FUNCTION_BLOCK "COM_Modbus_CMV96"	// FB 1709
TITLE = Serial communication (Modbus to CMV)
//  
//COPYRIGHT:    (C) 1997 BY  BUHLER LTD.
//                           CH-9240 UZWIL  SWITZERLAND
//
//PRODUCT:      GCS90S7
//
//TITLE:        Modbus Interface to CMV96
//
//-------------------------------------------------------------------------
//
//IDENT:        AUTHOR:             DEPT:                       DATE:
//
//FB1707.1.0    A.Egli              CT3                         29-Mar-2004
//              1st Release in S7
//
//-------------------------------------------------------------------------
//
//PURPOSE:      MANUAL : see [COMxxMAN]
//
//RESTRICTIONS: S7
//
//-------------------------------------------------------------------------
//
AUTHOR : EA
FAMILY : GCS90LL
NAME : CVMModb
VERSION : 1.0
VAR_INPUT
  InComID : WORD  := W#16#1000;
  InTick200ms : BOOL ;	// Tick is every 200ms for one scan high
END_VAR
VAR
  Spare4 : INT ;
  ParRetryCnt : INT  := 1;
  ParTimeOut : INT  := 30;	//Timebase 0.1 s
  Spare10 : INT ;
  Spare12 : INT ;
  Spare14 : INT ;
  InIdx : INT ;
  InOutRestartTime : INT  := 50;	//Timebase 0.1 s
  OutMaxIdx : INT  := 5;
  OutLenDataRecord : INT  := 70;
  Error : STRUCT
   LCAddr : INT ;
   Status : INT ;
   Count : INT ;
   StatusSnd : INT ;
   StatusRcv : INT ;
   Spare0 : INT ;
   Spare2 : INT ;
   Spare3 : INT ;
  END_STRUCT ;
  Telegram : STRUCT
   Idx : INT ;	// Index of actual communication job
   LCAddr : INT ;	// Index of LC which data are send
   TimeOut : INT ;	//
   Step : INT ;
   RetryCnt : INT ;
   spare3 : INT ;
   spare4 : INT ;
   spare5 : INT ;
   spare6 : INT ;
   spare7 : INT ;
  END_STRUCT ;
  CVM0 : STRUCT
   InRead : BOOL ;	// Command to read data
   OutComFault : BOOL ;
   InAddr : INT ;
   ActivePower : DINT ;
   ReactivePowerInductive : DINT ;
   ReactivePowerCapacitive : DINT ;
   VoltageL1 : DINT ;
   CurrentL1 : DINT ;
   VoltageL2 : DINT ;
   CurrentL2 : DINT ;
   VoltageL3 : DINT ;
   CurrentL3 : DINT ;
   Spare40 : DINT ;
   Spare44 : DINT ;
   Spare48 : DINT ;
   Spare52 : DINT ;
   Spare56 : DINT ;
   Spare58 : DINT ;
   RetryCnt : INT ;
   tmpParaNr : INT ;
   Spare68 : INT ;
  END_STRUCT ;
  CVM : ARRAY  [1 .. 5 ] OF STRUCT
   InRead : BOOL ;	// Command to read data
   OutComFault : BOOL ;
   InAddr : INT ;
   ActivePower : DINT ;
   ReactivePowerInductive : DINT ;
   ReactivePowerCapacitive : DINT ;
   VoltageL1 : DINT ;
   CurrentL1 : DINT ;
   VoltageL2 : DINT ;
   CurrentL2 : DINT ;
   VoltageL3 : DINT ;
   CurrentL3 : DINT ;
   Spare40 : DINT ;
   Spare44 : DINT ;
   Spare48 : DINT ;
   Spare52 : DINT ;
   Spare56 : DINT ;
   Spare58 : DINT ;
   RetryCnt : INT ;
   Spare66 : INT ;
   Spare68 : INT ;
  END_STRUCT ;
  DataSnd : STRUCT
   Ident : BYTE ;
   Func : BYTE ;
   Data : ARRAY  [1 .. 20 ] OF INT ;
  END_STRUCT ;
  DataRcv : ARRAY  [0 .. 30 ] OF DINT ;
  BSND : SFB 12;	//Data of CFB =====
  BRCV : SFB 13;	//Data of LC
END_VAR
VAR_TEMP
  tmpstoreAR2 : DINT ;
  tmpAddrLC : DINT ;
  tmpNo : INT ;
  tmpRestart : BOOL ;
  tmpNext : BOOL ;
  tmpLoop2 : BOOL ;
END_VAR
BEGIN
NETWORK
TITLE = Store
      TAR2  #tmpstoreAR2;
NETWORK
TITLE = Call Siemens SFB
      NOP   0;
//-Receive--
      SET;
      S     #BRCV.EN_R;
      L     #Telegram.Step;
      L     2;
      ==I;
      A     #BRCV.NDR;
      JC    rsJ1;
      BLD   16;
      =     L 17.0;
      L     DINO;
      T     LW 15;
      CDB;
      OPN   DI [LW 15];
      TAR2  LD 11;
      L     DBW [AR2,P#0.0];
      T     #BRCV.ID;
//-Send--
      L     W#16#1002;
      T     DIW [AR2,P#684.0];
      L     124;
      T     DIW [AR2,P#686.0];
      L     DBNO;
      T     DIW [AR2,P#688.0];
      +AR2  P#522.0;
      TAR2;
      LAR2  LD 11;
      T     DID [AR2,P#690.0];
      +AR2  P#672.0;
      UC    "SIEMENS_BRCV";
      LAR2  LD 11;
      CDB;
      BLD   17;
rsJ1: BLD   16;
      =     L 17.0;
      L     DINO;
      T     LW 15;
      CDB;
      OPN   DI [LW 15];
      TAR2  LD 11;
      L     DBW [AR2,P#0.0];
      T     #BSND.ID;
      L     W#16#1002;
      T     DIW [AR2,P#658.0];
      L     42;
      T     DIW [AR2,P#660.0];
      L     DBNO;
      T     DIW [AR2,P#662.0];
      +AR2  P#480.0;
      TAR2;
      LAR2  LD 11;
      T     DID [AR2,P#664.0];
      +AR2  P#646.0;
      UC    "SIEMENS_BSEND";
      LAR2  LD 11;
      CDB;
      BLD   17;
NETWORK
TITLE = Methode 0: Control Step "Init" 
//===================================================
//====Init if Restart PLC ========
      L     0;
      L     #InOutRestartTime;
      <I;
      =     #tmpRestart;
      AN    #tmpRestart;
      JC    InJ0;
      L     0;
      T     #Error.Count;
      R     #BRCV.NDR;
      R     #BRCV.ERROR;
// Set send and receive buffer 
      AN    #InTick200ms;	// 200ms second pulse
      JC    sav0;
      L     #InOutRestartTime;
      +     -2;
      T     #InOutRestartTime;
      BEU;
InJ0: NOP   0;
NETWORK
TITLE = Step: 0 to 3: Read Element Data
// read element data of active element 
// this part is done for Step 1,2,3
      SET;
      R     #tmpNext;
      R     #tmpLoop2;
S0:   L     1;
      L     #Telegram.Idx;
      >I;
      JC    S0Nx;
      L     #OutMaxIdx;
      >I;
      JC    S0Nx;
      L     #Telegram.Idx;
      +     -1;
      L     #OutLenDataRecord;
      SLD   3;
      *I;
      L     P##CVM;
      +D;
      T     #tmpAddrLC;
      LAR1  #tmpAddrLC;
      LAR2  P##CVM0;
      L     D [AR1,P#0.0];
      T     D [AR2,P#0.0];
      L     D [AR1,P#4.0];
      T     D [AR2,P#4.0];
      L     D [AR1,P#8.0];
      T     D [AR2,P#8.0];
      L     D [AR1,P#12.0];
      T     D [AR2,P#12.0];
      L     D [AR1,P#16.0];
      T     D [AR2,P#16.0];
      L     D [AR1,P#20.0];
      T     D [AR2,P#20.0];
      L     D [AR1,P#24.0];
      T     D [AR2,P#24.0];
      L     D [AR1,P#28.0];
      T     D [AR2,P#28.0];
      L     D [AR1,P#32.0];
      T     D [AR2,P#32.0];
      L     D [AR1,P#36.0];
      T     D [AR2,P#36.0];
      L     D [AR1,P#40.0];
      T     D [AR2,P#40.0];
      L     D [AR1,P#44.0];
      T     D [AR2,P#44.0];
      L     D [AR1,P#48.0];
      T     D [AR2,P#48.0];
      L     D [AR1,P#52.0];
      T     D [AR2,P#52.0];
      L     D [AR1,P#56.0];
      T     D [AR2,P#56.0];
      L     D [AR1,P#60.0];
      T     D [AR2,P#60.0];
      L     D [AR1,P#64.0];
      T     D [AR2,P#64.0];
      L     W [AR1,P#68.0];
      T     W [AR2,P#68.0];
      LAR2  #tmpstoreAR2;
NETWORK
TITLE = Methode 0:  Control: Step "Test queue"
      L     0;
      L     #Telegram.Step;
      <>I;
      JC    S1;
//Second Loop
      A     #tmpNext;
      A     #CVM0.InRead;
      JC    xxS1;	//-->Send telegram
//--Search next element ----
S0Nx: L     1;
      L     #Telegram.Idx;
      +     1;
      T     #Telegram.Idx;
      >I;
      JC    S0X1;
      L     #OutMaxIdx;
      <=I;
      JC    S0Do;
//--First Element ---
S0X1: L     1;
      T     #Telegram.Idx;	//Init with Index 1
      A     #tmpLoop2;
      BEC;
      S     #tmpLoop2;
//--read element data ---
S0Do: S     #tmpNext;
      JU    S0;
NETWORK
TITLE = Methode Control: Transition to Step 1: Prepare Send Telegram
//Call back element control before send
xxS1: L     0;
      T     #Telegram.TimeOut;
      L     #CVM0.RetryCnt;
      T     #Telegram.RetryCnt;
//Start Telegram
      L     #CVM0.InAddr;
      T     #Telegram.LCAddr;
      T     #DataSnd.Ident;
      L     4;
      T     #DataSnd.Func;
//1st Register
      L     #CVM0.tmpParaNr;
      L     0;
      <>I;
      JC    RdJ1;
      L     20;
RdJ1: T     #DataSnd.Data[1];
      T     #CVM0.tmpParaNr;
//1st Number of register to read
      L     #DataSnd.Data[2];
      L     22;
      ==I;
      L     24;
      JC    S1J1;
      TAK;
S1J1: T     #DataSnd.Data[2];	//Number of register to read
//length of send data
      L     8;
      T     #BSND.LEN;
//Set address send buffer
//Send Next step
      L     1;	//-->Emptying Buffer
      T     #Telegram.Step;
      L     0;
      T     #Telegram.TimeOut;
//Send Next step
NETWORK
TITLE = Methode Control: Step1: Emptying buffer
S1:   L     #Telegram.Step;
      L     1;
      <>I;
      JC    S2;
// Wait one scan
      L     #BSND.STATUS;
      L     0;
      <>I;
      O     #BRCV.NDR;
      O     #BRCV.ERROR;
      O     #BSND.REQ;
      O     #BSND.ERROR;
      O     #BSND.DONE;
      O     #BSND.REQ;
      R     #BRCV.NDR;
      R     #BRCV.ERROR;
      R     #BSND.REQ;
      R     #BSND.ERROR;
      R     #BSND.DONE;
      R     #BSND.REQ;
      JC    sav0;
//------------------------------------
//Next Step  : Send Telegramm
      L     2;
      T     #Telegram.Step;
      L     0;
      T     #Telegram.TimeOut;
      SET;
      S     #BSND.REQ;
NETWORK
TITLE = Methode Control: Step 2 :Send telegram 
S2:   L     #Telegram.Step;
      L     2;
      <>I;
      JC    S3;
// Test telegram done         
      A     #BRCV.NDR;
      A     #BSND.DONE;
      JC    xxS3;
// Test Nak         
      A     #BSND.ERROR;
      L     #BSND.STATUS;
      JC    NAK;
// Test TimeOut         
      AN    #InTick200ms;
      JC    sav0;
      L     #Telegram.TimeOut;
      +     2;
      T     #Telegram.TimeOut;
      L     #ParTimeOut;
      >I;
      L     128;	// TimeOut 
      JC    NAK;	//--> Time out 
      JU    sav0;
NETWORK
TITLE = Methode Control: Step 3 : Test answer telegram
xxS3: NOP   0;
//====================================================
//Compare telegram lenght with requestet answer length
      L     #DataSnd.Data[2];	//Number of register to read
      L     2;
      *I;
      L     #BRCV.LEN;
      <>I;
      L     140;
      JC    NAK;
//====================================================
//Store Data
      L     0;
      L     #DataSnd.Data[1];
      <>I;
      JC    AWJ1;
      L     #DataRcv[0];
      T     #CVM0.VoltageL1;
      L     #DataRcv[1];
      T     #CVM0.CurrentL1;
      L     #DataRcv[5];
      T     #CVM0.VoltageL2;
      L     #DataRcv[6];
      T     #CVM0.CurrentL2;
      L     #DataRcv[10];
      T     #CVM0.VoltageL3;
      L     #DataRcv[11];
      T     #CVM0.CurrentL3;
AWJ1: L     20;
      L     #DataSnd.Data[1];
      <>I;
      JC    AWJ9;
      L     #DataRcv[0];
      T     #CVM0.VoltageL3;
      L     #DataRcv[1];
      T     #CVM0.CurrentL3;
      L     #DataRcv[5];
      T     #CVM0.ActivePower;
      L     #DataRcv[6];
      T     #CVM0.ReactivePowerInductive;
      L     #DataRcv[7];
      T     #CVM0.ReactivePowerCapacitive;
AWJ9: SET;
      R     #CVM0.OutComFault;
NETWORK
TITLE = Methode Control: Step 3: Init for next Telegram
S3:   L     0;
      T     #CVM0.RetryCnt;
S3rt: SET;
      R     #BRCV.NDR;
      R     #BRCV.ERROR;
      R     #BSND.DONE;
      R     #BSND.ERROR;
//--Step 0 -----
      L     0;
      T     #Telegram.Step;
      JU    sav0;
NETWORK
TITLE = Methode Control: NAK 
///
//Error send 
NAK:  T     #Error.Status;
      L     #Telegram.LCAddr;
      T     #Error.LCAddr;
      L     #Error.Count;
      +     1;
      T     #Error.Count;
      L     #BSND.STATUS;
      T     #Error.StatusSnd;
      L     #BRCV.STATUS;
      T     #Error.StatusRcv;
      L     #ParRetryCnt;
      L     #CVM0.RetryCnt;
      >I;	//--> Retry after fault 
      O     #tmpRestart;	//--> Retry during restart
      JC    naRt;	//--> Retry after fault 
      L     0;
      T     #CVM0.RetryCnt;
      S     #CVM0.OutComFault;
      JU    S3;
naRt: L     #CVM0.RetryCnt;
      +     1;
      T     #CVM0.RetryCnt;
      JU    S3rt;
NETWORK
TITLE = Methode 2: Store element data 
sav0: L     1;
      L     #Telegram.Idx;
      >I;
      BEC;
      L     #OutMaxIdx;
      >I;
      BEC;
      L     #Telegram.Idx;
      +     -1;
      L     #OutLenDataRecord;
      SLD   3;
      *I;
      L     P##CVM;
      +D;
      T     #tmpAddrLC;
      LAR1  P##CVM0;
      LAR2  #tmpAddrLC;
      L     D [AR1,P#0.0];
      T     D [AR2,P#0.0];
      L     D [AR1,P#4.0];
      T     D [AR2,P#4.0];
      L     D [AR1,P#8.0];
      T     D [AR2,P#8.0];
      L     D [AR1,P#12.0];
      T     D [AR2,P#12.0];
      L     D [AR1,P#16.0];
      T     D [AR2,P#16.0];
      L     D [AR1,P#20.0];
      T     D [AR2,P#20.0];
      L     D [AR1,P#24.0];
      T     D [AR2,P#24.0];
      L     D [AR1,P#28.0];
      T     D [AR2,P#28.0];
      L     D [AR1,P#32.0];
      T     D [AR2,P#32.0];
      L     D [AR1,P#36.0];
      T     D [AR2,P#36.0];
      L     D [AR1,P#40.0];
      T     D [AR2,P#40.0];
      L     D [AR1,P#44.0];
      T     D [AR2,P#44.0];
      L     D [AR1,P#48.0];
      T     D [AR2,P#48.0];
      L     D [AR1,P#52.0];
      T     D [AR2,P#52.0];
      L     D [AR1,P#56.0];
      T     D [AR2,P#56.0];
      L     D [AR1,P#60.0];
      T     D [AR2,P#60.0];
      L     D [AR1,P#64.0];
      T     D [AR2,P#64.0];
      L     W [AR1,P#68.0];
      T     W [AR2,P#68.0];
      LAR2  #tmpstoreAR2;
END_FUNCTION_BLOCK

FUNCTION_BLOCK "SSA_EL_Sampler_RFID"	// FB 1714
TITLE = Lesen/Schreiben 2k bit / Profibus DP
//COPYRIGHT:    (C) 2006  BUHLER AG, CH-9240 UZWIL, SWITZERLAND
//
//PRODUCT:      GCS7R2
//
//TITLE:        RFID Baumer
//
//REVISION:     20
//-------------------------------------------------------------------------
//
//IDENT:        AUTHOR:             DEPT:                       DATE:
//FB1714.1.0    A. Egli             CT3                         12-Sep-2007
//              #FromBuhler.InSimulation to read/write process immage
//FB1714.1.0    A. Egli             CT3                         19-Mar-2007
//              New Release R2
//
//-------------------------------------------------------------------------
//
//PURPOSE:      MANUAL : see [SSW-EL-Sampler_MAN_en]
//              This FB is a copy of original communication block FB102 of 
//              Baumer. 
//
//              Modification of BUHLER:
//              - Move all IN and OUT signal to the area STAT.
//              - Add all data of the global DB of Baumer into are STAT
//                (STAT:IN,STAT:OUT)
//                The structur IN must start at Byte 0
//                The structur OUT must start at Byte 204
//                This because Baumer uses the absoulte address of thes tags
//             - Add interface to BUHLER elements
//               (FromBuhler, ToBuhler)  
//              
//
//RESTRICTIONS: S7
//
//-------------------------------------------------------------------------
//
AUTHOR : ZIEGERT
FAMILY : BAUMER
NAME : RFID
VERSION : 1.1
VAR
  IN : STRUCT 	//Read buffer
   CONTROL1 : WORD ;	//Commando / # antenne
   CONTROL2 : WORD ;	//State of central unit / # pages
   CONTROL3 : WORD ;	//# datablocks / Actual datablock
   CONTROL4 : WORD ;	//Length of datablock / Controlbyte
   PAGE16 : DWORD ;	//Nutzdaten 1 Input
   PAGE17 : DWORD ;	//Nutzdaten 2 Input
   PAGE18 : DWORD ;	//Nutzdaten 3 Input
   PAGE19 : DWORD ;	//Nutzdaten 4 Input
   PAGE20 : DWORD ;	//Nutzdaten 5 Input
   PAGE21 : DWORD ;	//Nutzdaten 6 Input
   PAGE22 : DWORD ;	//Nutzdaten 7 Input
   PAGE23 : DWORD ;	//Nutzdaten 8 Input
   PAGE24 : DWORD ;	//Nutzdaten 9 Input
   PAGE25 : DWORD ;	//Nutzdaten 10 Input
   PAGE26 : DWORD ;	//Nutzdaten 11 Input
   PAGE27 : DWORD ;	//Nutzdaten 12 Input
   PAGE28 : DWORD ;	//Nutzdaten 13 Input
   PAGE29 : DWORD ;	//Nutzdaten 14 Input
   PAGE30 : DWORD ;	//Nutzdaten 15 Input
   PAGE31 : DWORD ;	//Nutzdaten 16 Input
   PAGE32 : DWORD ;	//Nutzdaten 17 Input
   PAGE33 : DWORD ;	//Nutzdaten 18 Input
   PAGE34 : DWORD ;	//Nutzdaten 19 Input
   PAGE35 : DWORD ;	//Nutzdaten 20 Input
   PAGE36 : DWORD ;	//Nutzdaten 21 Input
   PAGE37 : DWORD ;	//Nutzdaten 22 Input
   PAGE38 : DWORD ;	//Nutzdaten 23 Input
   PAGE39 : DWORD ;	//Nutzdaten 24 Input
   PAGE40 : DWORD ;	//Nutzdaten 25 Input
   PAGE41 : DWORD ;	//Nutzdaten 26 Input
   PAGE42 : DWORD ;	//Nutzdaten 27 Input
   PAGE43 : DWORD ;	//Nutzdaten 28 Input
   PAGE44 : DWORD ;	//Nutzdaten 29 Input
   PAGE45 : DWORD ;	//Nutzdaten 30 Input
   PAGE46 : DWORD ;	//Nutzdaten 31 Input
   PAGE47 : DWORD ;	//Nutzdaten 32 Input
   PAGE48 : DWORD ;	//Nutzdaten 33 Input
   PAGE49 : DWORD ;	//Nutzdaten 34 Input
   PAGE50 : DWORD ;	//Nutzdaten 35 Input
   PAGE51 : DWORD ;	//Nutzdaten 36 Input
   PAGE52 : DWORD ;	//Nutzdaten 37 Input
   PAGE53 : DWORD ;	//Nutzdaten 38 Input
   PAGE54 : DWORD ;	//Nutzdaten 39 Input
   PAGE55 : DWORD ;	//Nutzdaten 40 Input
   PAGE56 : DWORD ;	//Nutzdaten 41 Input
   PAGE57 : DWORD ;	//Nutzdaten 42 Input
   PAGE58 : DWORD ;	//Nutzdaten 43 Input
   PAGE59 : DWORD ;	//Nutzdaten 44 Input
   PAGE60 : DWORD ;	//Nutzdaten 45 Input
   PAGE61 : DWORD ;	//Nutzdaten 46 Input
   PAGE62 : DWORD ;	//Nutzdaten 47 Input
   PAGE63 : DWORD ;	//Nutzdaten 48 Input
   Spare : DWORD ;	//spare
  END_STRUCT ;
  OUT : STRUCT 	//Write buffer
   CONTROL1 : WORD ;	//Commando / # antenne
   CONTROL2 : WORD ;	//Startpage / # pages
   CONTROL3 : WORD ;	//# datablocks / Actual datablock
   CONTROL4 : WORD ;	//Length of datablock / Controlbyte
   PAGE16 : DWORD ;	//Nutzdaten 1 Output
   PAGE17 : DWORD ;	//Nutzdaten 2 Output
   PAGE18 : DWORD ;	//Nutzdaten 3 Output
   PAGE19 : DWORD ;	//Nutzdaten 4 Output
   PAGE20 : DWORD ;	//Nutzdaten 5 Output
   PAGE21 : DWORD ;	//Nutzdaten 6 Output
   PAGE22 : DWORD ;	//Nutzdaten 7 Output
   PAGE23 : DWORD ;	//Nutzdaten 8 Output
   PAGE24 : DWORD ;	//Nutzdaten 9 Output
   PAGE25 : DWORD ;	//Nutzdaten 10 Output
   PAGE26 : DWORD ;	//Nutzdaten 11 Output
   PAGE27 : DWORD ;	//Nutzdaten 12 Output
   PAGE28 : DWORD ;	//Nutzdaten 13 Output
   PAGE29 : DWORD ;	//Nutzdaten 14 Output
   PAGE30 : DWORD ;	//Nutzdaten 15 Output
   PAGE31 : DWORD ;	//Nutzdaten 16 Output
   PAGE32 : DWORD ;	//Nutzdaten 17 Output
   PAGE33 : DWORD ;	//Nutzdaten 18 Output
   PAGE34 : DWORD ;	//Nutzdaten 19 Output
   PAGE35 : DWORD ;	//Nutzdaten 20 Output
   PAGE36 : DWORD ;	//Nutzdaten 21 Output
   PAGE37 : DWORD ;	//Nutzdaten 22 Output
   PAGE38 : DWORD ;	//Nutzdaten 23 Output
   PAGE39 : DWORD ;	//Nutzdaten 24 Output
   PAGE40 : DWORD ;	//Nutzdaten 25 Output
   PAGE41 : DWORD ;	//Nutzdaten 26 Output
   PAGE42 : DWORD ;	//Nutzdaten 27 Output
   PAGE43 : DWORD ;	//Nutzdaten 28 Output
   PAGE44 : DWORD ;	//Nutzdaten 29 Output
   PAGE45 : DWORD ;	//Nutzdaten 30 Output
   PAGE46 : DWORD ;	//Nutzdaten 31 Output
   PAGE47 : DWORD ;	//Nutzdaten 32 Output
   PAGE48 : DWORD ;	//Nutzdaten 33 Output
   PAGE49 : DWORD ;	//Nutzdaten 34 Output
   PAGE50 : DWORD ;	//Nutzdaten 35 Output
   PAGE51 : DWORD ;	//Nutzdaten 36 Output
   PAGE52 : DWORD ;	//Nutzdaten 37 Output
   PAGE53 : DWORD ;	//Nutzdaten 38 Output
   PAGE54 : DWORD ;	//Nutzdaten 39 Output
   PAGE55 : DWORD ;	//Nutzdaten 40 Output
   PAGE56 : DWORD ;	//Nutzdaten 41 Output
   PAGE57 : DWORD ;	//Nutzdaten 42 Output
   PAGE58 : DWORD ;	//Nutzdaten 43 Output
   PAGE59 : DWORD ;	//Nutzdaten 44 Output
   PAGE60 : DWORD ;	//Nutzdaten 45 Output
   PAGE61 : DWORD ;	//Nutzdaten 46 Output
   PAGE62 : DWORD ;	//Nutzdaten 47 Output
   PAGE63 : DWORD ;	//Nutzdaten 48 Output
   PAGE64 : DWORD ;	//Nutzdaten 49 Output
  END_STRUCT ;
  spare408 : BOOL ;
  FromBuhler : STRUCT
   BottleInPosition : BOOL ;	//LS tells that a bottle is in position
   StBottleChange : BOOL ;	//Bottle change is avtive
   CmdFaultReset : BOOL ;	//Reset Retry Counter
   ParTag2KB : BOOL ;	//1=2kByte  , 0=256Byte
   InSimulation : BOOL ;	//1=Connected to IOSimuli
   ParByteNo : INT ;	//1st Byte of ID
   spare1 : INT ;
   spare2 : INT ;
   spare3 : INT ;
  END_STRUCT ;
  ToBuhler : STRUCT
   OutReadingFault : BOOL ;
   RFIDJobRunning : BOOL ;	//Data for user
   EdgeBottleInPossition : BOOL ;	//Data for user
   RFIDStartReading : BOOL ;	//Data for user
   OutEdgeBreak : BOOL ;
   OutEdgeRW_End : BOOL ;
   OutPulseRW_End : BOOL ;
   OutRFIDBusy : BOOL ;
   OutEdgeRFIDIdling : BOOL ;
   OutPulseRFIDIdling : BOOL ;
   OutRFIDIdling : BOOL ;
   OutTimeOut : INT ;
   OutTagNoAct : DINT ;
   OutDelayBrake : INT ;
   OutRetryCounter : INT ;
   spare1 : INT ;
   spare2 : INT ;
   spare3 : INT ;
   spare4 : INT ;
   spare5 : INT ;
  END_STRUCT ;
  START_RW : BOOL ;	//Start read/write Auftrag
  BREAK : BOOL ;	//Break read/write
  READ : BOOL ;	//Commando read
  WRITE : BOOL ;	//Commando write
  POLL : BOOL ;	//Mode poll
  AUTO : BOOL ;	//Mode automatic
  CONT : BOOL ;	//Mode continues
  ANT : INT ;	//Nr. der Antenne (Wert 0-2)
  STARTP : INT ;	//Startpage (Wert >=16, <=48)
  ANZP : INT ;	//Anzahl Page Extern (Wert = 1-48)
  EA_or_PW : INT ;	//Vorwahl Adressbereich E/A oder PW, (Wert 0 = E/A Wert 1 = PW)
  EADR : INT ;	//Anfangsaddresse Eingänge (Daten vom slave)
  AADR : INT ;	//Anfangsaddresse Ausgänge (Daten vom slave)
  T_MS : INT ;	//Zeitwert für Time out
  STATE_HW : BYTE ;	//Status des OIS-L Controller's (read/write system)
  STATE_HS : BYTE ;	//Status handshake
  RW_END : BOOL ;	//Read/Write Ende
  TIMEOUT : BOOL ;	//Timeout
  PARA : BOOL ;	//Parameterfehler
  FLT : BOOL ;	//Sammelfehler
  HW_FLT : BOOL ;	//Hardware Fehler OIS-L Controller
  P_start_rw : BOOL ;	//Flanke 'START_RW'
  E_start_rw : BOOL ;	//Hilfsmerker 'START_RW'
  RW_act : BOOL ;	//Auftrag gestartet
  P_rw_end : BOOL ;	//Pos. Flanke Lese/schreiben ende
  E_rw_end : BOOL ;	//Enable Flanke Lesen/schreiben Ende
  ANZP_SAVE : INT ;	//Pageanzahl sichern
  anz_page : INT ;	//Anzahl Page intern (wert = 0-15)
  anz_blocks : INT ;	//# Anzahl Datenblocks
  act_block : INT ;	//# Write: Aktueller Datenblock
  rest_bytes : INT ;	//# Anzahl Restbyte's die ggelesen/geschrieben werden
  anz_bytes : INT ;	//# Anzahl Byt's gesamt
  rcv_blocks : INT ;	//# Aktueller Blockzeiger
  P_OIS_new_data : BOOL ;	//# Read: Flanke start neue Daten Lesen
  E_OIS_new_data : BOOL ;	//# Read: Hilfsmerker: neue Daten Lesen
  P_OIS_data_rcv : BOOL ;	//# Write: Flanke start neue Daten Schreiben
  E_OIS_data_rcv : BOOL ;	//# Write: Hilfsmerker: neue Date Schreiben
  RD : BOOL ;	//# Read: Start Daten Lesen
  RD_no_active : BOOL ;	//# Read/Write: Daten Lesen/Schreiben nicht active
  WR : BOOL ;	//# Write: Start Daten Schreiben
  pointer_dest : DWORD ;	//Pointer Hilfsregister zum zwischenspeichern des Zeigers
  Pointer_buffer : DWORD ;	//Pointer aktueller Zeiger auf Daten/Adressbereich
  s_pointer_set : BOOL ;	//Pointer_buffer gesetzt
  S_break : BOOL ;	//positive Flanke Breakbefehl gestartet
  E_break : BOOL ;	//Flankenmerker Break
  N_break : BOOL ;	//negative Flanke nach S_break, Break an OIS-L senden
  S_poll : BOOL ;	//Mode poll angewählt
  E_en_poll : BOOL ;	//Hilfsmerker poll angewählt
  S_auto : BOOL ;	//Mode auto angewählt
  E_en_auto : BOOL ;	//Hilfsmerker auto angewählt
  S_cont : BOOL ;	//Mode cont angewählt
  E_en_cont : BOOL ;	//Hilfsmerker cont angewählt
  anz_loop : INT ;	//# Read/Write: Anzahl der errechneten loop's
  Loop : INT ;	//Schleife für mehrfachse Lesen (Wert 0-2)
  S_loop : BOOL ;	//Schleifenmerker (1 wenn mehr als 16 Page gelesen werden sollen)
  S_Data_1 : BOOL ;	//Berechnung für Startpage und Anzahl Page durchgeführt
  E_en_Bussy : BOOL ;	//Auftrag gestartet
  P_en_DATA : BOOL ;	//Hilfsmerker pos.Flanke: neue daten vom Slave vorhanden
  N_en_DATA : BOOL ;	//Hilfsmerker neg.Flanke: neue daten vom Slave vorhanden
  E_en_DATA : BOOL ;	//Flanke neue Daten vom Slave vorhanden
  adb_dbn : BOOL ;	//# Read/Write: Controll In ADB = DBN
  errCDO : BOOL ;	//Fehler
  errMOD : BOOL ;	//Fehler Mode Read/Write (beide angewählt)
  errANT : BOOL ;	//Fehler Nr. der Antenne (darf nur 1 oder 2 sein)
  errSTARTP : BOOL ;	//Fehler Startpage (min Wert 16, max Wert 63)
  errANZP : BOOL ;	//Fehler Anzahl Page {min Wert 1, max Wert 48 (cont mode max 16)}
  errDATA : BOOL ;	//Fehler Datenlänge und Controllbit CTL.0 und CTL.2
  E_CTL_7_out : BOOL ;	//Flankenmerker CTL.7 out
  s_timeout : BOOL ;	//Start Timeout bei CLT(out)<> CLT(in)
  s_daten_ok : BOOL ;	//Daten liegen auf den Ausgängen (write)
  s_next_block : BOOL ;	//Daten an oil-s, nächsten Block senden
  dummy : BOOL ;	//Schmiermerker
  result : INT ;	//Hilfsregister: Check Anzahl page
  rest_page : INT ;	//Register: dient zum zwischenspeichern der neu ermittelten Pageanzahl
  Pointer_input : DWORD ;	//Pointer input: Zeiger auf Eingangsbereich
  Pointer_output : DWORD ;	//Pointer output: Zeiger auf Ausgangsbereich
  RD_loop_counter : INT ;	//#Read/Write: Schleifenzähler beim Lesen und Schreiben
END_VAR
VAR_TEMP
  tmpDB : INT ;
  tmpTOut : INT ;
END_VAR
BEGIN
NETWORK
TITLE =
//Dieser FB ist die Schnittstelle für das Lesen und Schreiben von 2k Tag's über 
//den Profibus DP vom oder zum OIS-L Kontroller.
//Folgende Funktionen können mit dem FB realiesiert werden:
//Lesen von 48 Page im Poll und Auto Mode
//Lesen von 16 Page im Cont Mode
//Schreiben von 48 Page im Poll und Auto Mode
//Das Schreiben im Cont Mode ist nicht möglich.
//--------------------------------------------------------------------------------
//Die Beschreibung der einzelnen Modis ist dem Benutzerhandbuch für den OIS-L 
//Kontroller zu entnehmen.
//--------------------------------------------------------------------------------
//Datenstruktur im _DB
//DB102--------------------
//DBW0  Comando/Antenne                      [IN]
//DBW2  Status/AnzPage                       [IN]
//DBW4  AnzDatenblöcke/Nr.Akt.Datenblock     [IN]
//DBW6  Datenlänge/Controllbyte              [IN]
//DD8-DD196  Daten Page 16-63                [IN]
//
//DBW204 Comando/Antenne                     [OUT]
//DBW206 Status/AnzPage                      [OUT]
//DBW208 AnzDatenblöcke/Nr.Akt.Datenblock    [OUT]
//DBW210 Datenlänge/Controllbyte             [OUT]
//DD212-DD400 Daten Page 16-63               [OUT]
//
//Achtung: Der Datenbereich für Daten von Antenne 1 und Daten von Antenne 2 sind 
//identisch.  Alternativ können auch bei einem Mehrfachaufruf zwei Datenbausteine 
//eingesetzt werden, in denen die Tag-Daten abgespeichert werden.
//Bei Mehrfachaufrufen ist darauf zu achten, das bevor der FB durchlaufen wird 
//ein Break Befehl durchgeführt wird.
//
//Weiterhin ist darauf zu achten, dass die FB's gegeneinander Verriegelt werden.
//Ein Möglichkeit ist es durch die Anwahl der Antennen den EN Eingang der FB's zu 
//selktieren und das RD_End Signal als Quittierung zu benutzen.
//
//Continius-Mode:
//Nach einem Break-Befehl während des Continius-Mode muß erneut ein Startbefehl 
//abgesetzt werden um das Lesen zu starten:
//
//Zusätzlich benötig der FB noch einen Instanz DB, der beim Aufruf des FB's 
//eingetragen werden muß. Es ist nicht empfehlenswert den FB105 in eine 
//Multiinstanz abzuändern.
//
//Parameterbeschreibung:
//---------EINGÄNGE----------
//EN       [Bool]     Enable muß auf Logisch 1 sein.
//_DB      [Bloch_DB] Datenbaustein der die Tagdaten sowie Status-und Steuerwort  
//                    enthält.
//START_RD [Bool]     Daten lesen start im Poll- und Auto-Mode.
//BREAK    [Bool]     Hi aktiv, setzt den IBS-OISL-Protokollkoppler
//POLL     [Bool]     Hi aktiv Pollmodus.
//AUTO     [Bool]     Hi aktiv Automatikmodus.
//CONT     [Bool]     Hi aktiv Continiusmode.
//READ     [Bool]     Hi aktiv selektiert den Lesevorgang
//WRITE    [Bool]     Hi aktiv selektiert den Schreibvorgang 
//ANT      [Int]      Wert 1 oder 2 aktiviert den Anteneneingang 1 oder 2.
//STARTP   [INT]      Wert 16-63 Vorwahl der Page, ab der Daten gelesen oder
//                    beschrieben werden sollen
//ANZP     [INT]      Wert 1-48 Anzahl Page's die gelesen oder beschrieben werden 
//                    sollen {max. 48 Page's können gelesen oder beschrieben 
//                    werden, im cont Mode ist das lesen auf 16 Page reduziert}.
//EA_or_PW [Int]      Ermöglicht die Anpassung des Einganmgsbereichs Wert 0=EA,   
//                    Wert 1=PW (PW = Peripheriebereich)
//EADR     [Int]      Wert je nach parametrierten Eingangsbereich Profibus/S7.
//AADR     [Int]      Wert je nach parametrierten Eingangsbereich Profibus/S7.
//T_OUT    [Timer]    S7 Zeit (z.B. T10) Überwachung der Lesefunktion im 
//                    AUTO-CONT-Mode.
//T_OUT_MS [S5Time]   Zeitbereich von T_OUT (z.B. S5T#10s).
//
//---------AUSGÄNGE----------
//ENO      [Bool]     Logisch 1 wenn EN Logisch 1 ist.
//STATE_HW [Byte]     Status und Errocode des OISL-Protokollkoppler.
//State_HS [Byte]     Status Controllbyts des OISL-Protokollkoppler.
//RD_END   [Bool]     Hi aktiv, Lese/Schreib-Auftrag beendet.
//TIMEOUT  [Bool]     Hi aktiv, Zeitüberschreitung beim lesen (kein Tag im        
//                    Antennenbereich).
//PARA     [Bool]     Hi aktiv, Falsche Parameter an den Eingängen POLL, AUTO,CONT
//                    oder ANT.
//FLT      [Bool]     Hi aktiv, Summenfehler.
//
//Beschreibung zum Ablauf:
//Liegt an den Eingängen (Poll, Auto, Cont oder Antenne) kein Singnal wird der 
//Ausgang PARA und FTL gesetzt und zum Ende verzweigt.
//Nachdem ein Modus gewählt wurde kann das Lesen/Schreiben der Daten mit START_RD 
//eingeleitet werden. Ein beschreiben der Tag's im Continus-Mode ist nicht 
//möglich.
//Wurde ein Modus vorgewählt und das Lesen der Daten gestartet, sollte bei einem 
//wechsel des Modus immer ein Reset Buffer durchgeführt werden.
//Im Auto/Cont Mode ist die Zeitüberwachung aktiv im Poll Mode nicht.
//Im Cont_Mode führt eine Pageanzahl >16 zum setzten des Fehlerausgangs.
//Ein Break-Befehl kann nur bei eindeutiger Parametrierung am Eingang 
//durchgeführt werden.
//Wird als StartPage 0 und AnzahlPage 1 vorgegeben, wird die TAG ID ausgelesen. 
//
NETWORK
TITLE = [1.0] öffen _DB 
      L     DINO;
      T     #tmpDB;
      OPN   DB [#tmpDB];
NETWORK
TITLE = [1.0] BUZ: Command from Buhler to Baumer RFID (Part 1)
      NOP   0;
//-Initialize ---
      AN    DIX 442.2;
      S     DIX 442.2;
      S     DIX 442.1;
// 
//-Reading---
      A     DIX 410.0;
      AN    DIX 410.2;
      FP    DIX 420.2;
      S     DIX 420.3;
// 
      A     DIX 420.3;
      AN    DIX 420.7;
      A     DIX 421.2;
      AN    DIX 442.1;
      S     DIX 442.0;
//WinTrend      L     S5T#150MS
//WinTrend      SV    T    200
//WinTrend      U     T    200
//WinTrend      =     M   1400.0
// 
      O     DIX 410.1;
      R     DIX 420.3;
// 
//-Set default data---
      SET;
      R     DIX 442.3;
      S     DIX 442.4;
      R     DIX 442.5;
      R     DIX 442.6;
      L     0;	//[1.1]
      A     DIX 410.4;	//[1.1]
      JC    SiEA;	//[1.1]
      L     1;
SiEA: T     DIW 450;
      L     1;
      T     DIW 444;
      L     0;
      T     DIW 446;
      L     1;
      T     DIW 448;
      L     DIW 412;
      T     DIW 452;
      L     DIW 412;
      T     DIW 454;
      L     2000;
      T     DIW 456;
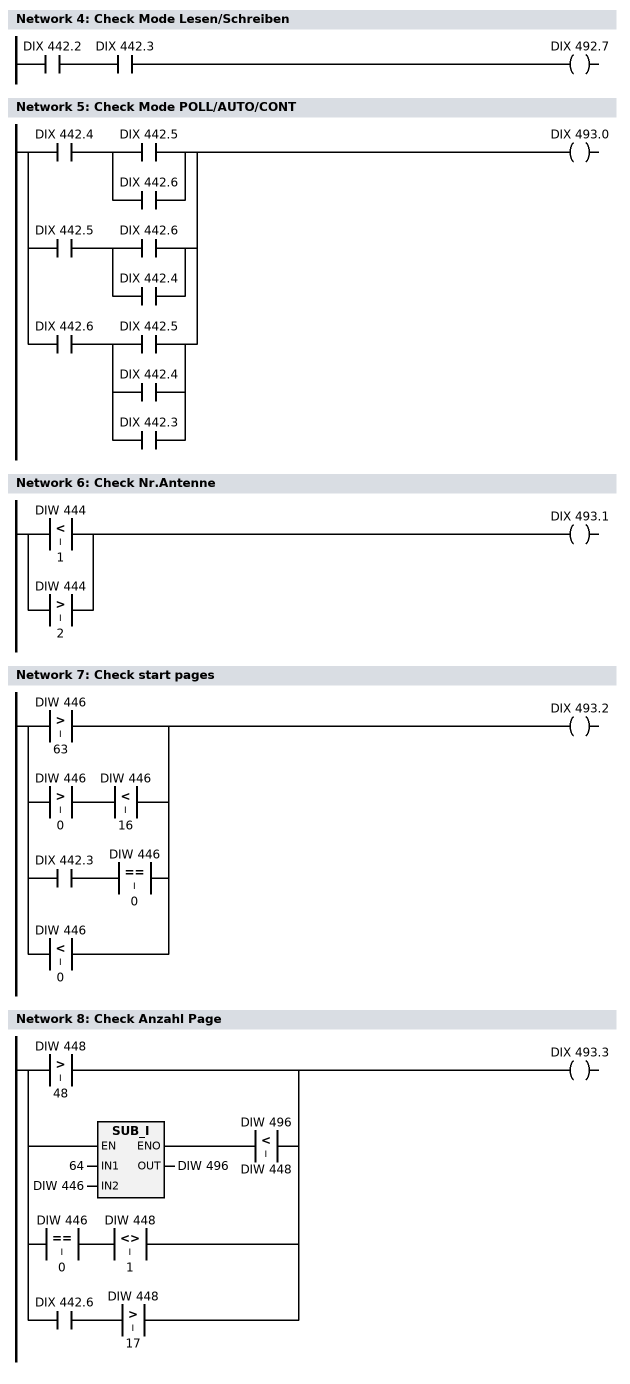
NETWORK
TITLE = Check Mode Lesen/Schreiben
      A     DIX 442.2;
      A     DIX 442.3;
      =     DIX 492.7;
NETWORK
TITLE = Check Mode POLL/AUTO/CONT
      A     DIX 442.4;
      A(;
      O     DIX 442.5;
      O     DIX 442.6;
      );
      O;
      A     DIX 442.5;
      A(;
      O     DIX 442.6;
      O     DIX 442.4;
      );
      O;
      A     DIX 442.6;
      A(;
      O     DIX 442.5;
      O     DIX 442.4;
      O     DIX 442.3;
      );
      =     DIX 493.0;
NETWORK
TITLE = Check Nr.Antenne
      O(;
      L     DIW 444;
      L     1;
      <I;
      );
      O(;
      L     DIW 444;
      L     2;
      >I;
      );
      =     DIX 493.1;
NETWORK
TITLE = Check start pages
      O(;
      L     DIW 446;
      L     63;
      >I;
      );
      O;
      A(;
      L     DIW 446;
      L     0;
      >I;
      );
      A(;
      L     DIW 446;
      L     16;
      <I;
      );
      O;
      A     DIX 442.3;
      A(;
      L     DIW 446;
      L     0;
      ==I;
      );
      O(;
      L     DIW 446;
      L     0;
      <I;
      );
      =     DIX 493.2;
NETWORK
TITLE = Check Anzahl Page
      O(;
      L     DIW 448;
      L     48;
      >I;
      );
      O(;
      A(;
      L     64;
      L     DIW 446;
      -I;
      T     DIW 496;
      AN    OV;
      SAVE;
      CLR;
      A     BR;
      );
      A(;
      L     DIW 496;
      L     DIW 448;
      <I;
      );
      );
      O;
      A(;
      L     DIW 446;
      L     0;
      ==I;
      );
      A(;
      L     DIW 448;
      L     1;
      <>I;
      );
      O;
      A     DIX 442.6;
      A(;
      L     DIW 448;
      L     17;
      >I;
      );
      =     DIX 493.3;
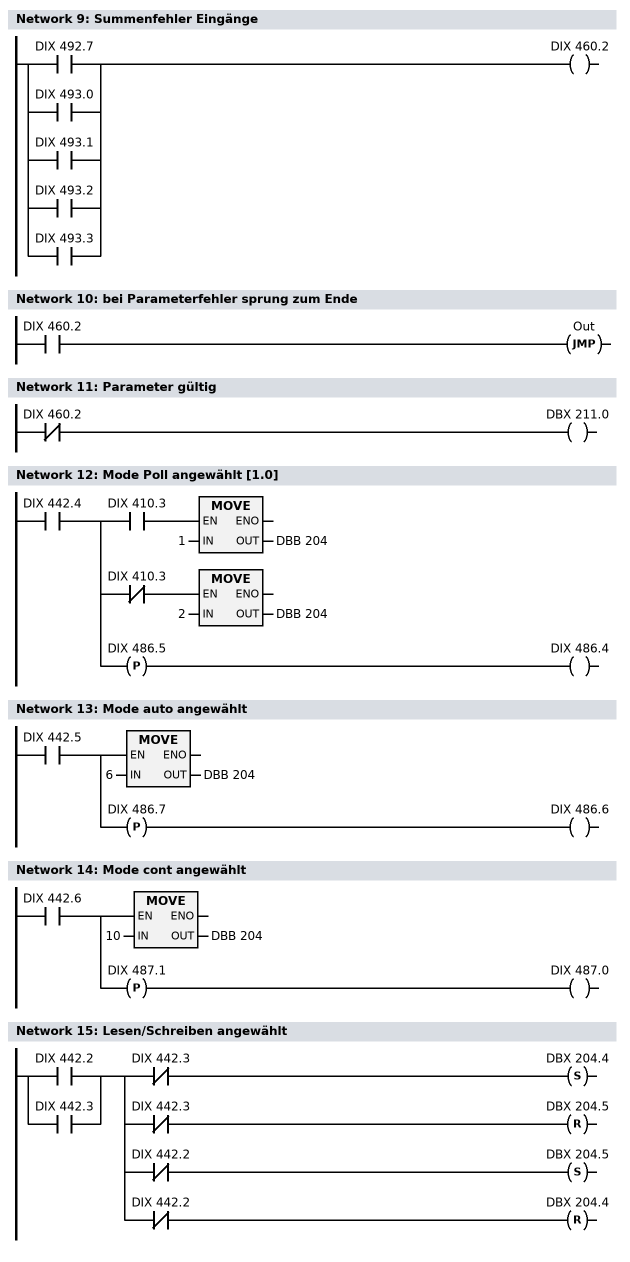
NETWORK
TITLE = Summenfehler Eingänge
      O     DIX 492.7;
      O     DIX 493.0;
      O     DIX 493.1;
      O     DIX 493.2;
      O     DIX 493.3;
      =     DIX 460.2;
NETWORK
TITLE = bei Parameterfehler sprung zum Ende
      A     DIX 460.2;
      JC    Out;
NETWORK
TITLE = Parameter gültig
//CTL.0=1
      AN    DIX 460.2;
      =     DBX 211.0;
NETWORK
TITLE = Mode Poll angewählt [1.0]
//Modus: Bitmuster
//BIT:  7654 32 10
//      0000 00 01 -->POLL 2K Tag 1  ¦¦ 0000 00 10 -->POLL 256Bit Tag 2
//      0000 01 01 -->AUTO 2K Tag 5  ¦¦ 0000 01 10 -->AUTO 256Bit Tag 6
//      0000 10 01 -->CONT 2K Tag 9  ¦¦ 0000 10 10 -->CONT 256Bit Tag 10
//für READ/WRITE wird das 4/5 Bit seperat gesetzt!
      A     DIX 442.4;
      =     L 4.0;	//Poll mode
      A     L 4.0;
      A     DIX 410.3;
      JNB   _001;
      L     1;
      T     DBB 204;
_001: NOP   0;
      A     L 4.0;
      AN    DIX 410.3;
      JNB   _002;
      L     2;
      T     DBB 204;
_002: NOP   0;
      A     L 4.0;
      FP    DIX 486.5;
      =     DIX 486.4;
NETWORK
TITLE = Mode auto angewählt
//...siehe Poll-Modus Netzwerk 10
      A     DIX 442.5;	//Continouse mode
      =     L 4.0;
      A     L 4.0;
      JNB   _003;
      L     6;
      T     DBB 204;
_003: NOP   0;
      A     L 4.0;
      FP    DIX 486.7;
      =     DIX 486.6;
NETWORK
TITLE = Mode cont angewählt
//...siehe Poll-Modus Netzwerk 10
      A     DIX 442.6;
      =     L 4.0;
      A     L 4.0;
      JNB   _007;
      L     10;
      T     DBB 204;
_007: NOP   0;
      A     L 4.0;
      FP    DIX 487.1;
      =     DIX 487.0;
NETWORK
TITLE = Lesen/Schreiben angewählt
      O     DIX 442.2;
      O     DIX 442.3;
      =     L 4.0;
      A     L 4.0;
      AN    DIX 442.3;
      S     DBX 204.4;
      A     L 4.0;
      AN    DIX 442.3;
      R     DBX 204.5;
      A     L 4.0;
      AN    DIX 442.2;
      S     DBX 204.5;
      A     L 4.0;
      AN    DIX 442.2;
      R     DBX 204.4;
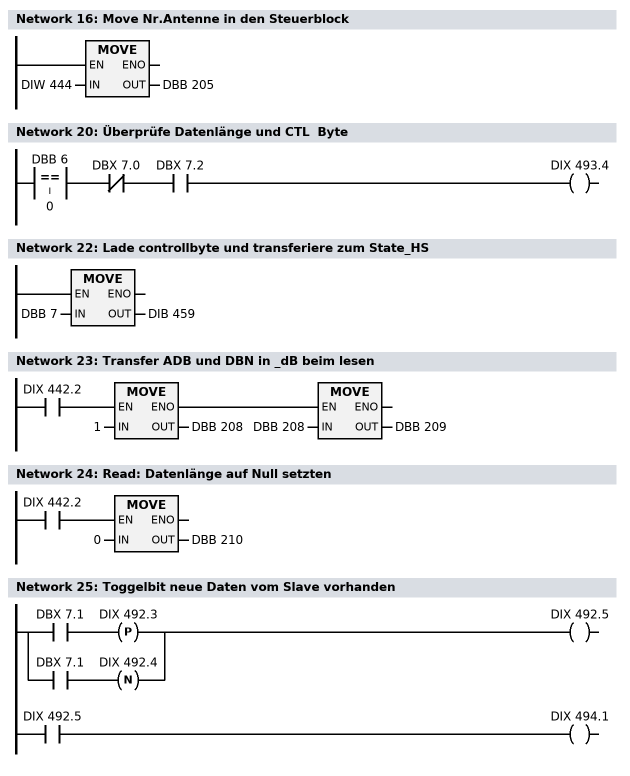
NETWORK
TITLE = Move Nr.Antenne in den Steuerblock
//Der Wert für Antenne 1 ist 1 und für Antenne 2 ist 2
      L     DIW 444;
      T     DBB 205;
      NOP   0;
NETWORK
TITLE = Berechnung und übertragen von Startpage und Anzahl Page
//6 pages (each 4 bytes) = 24 bytes = 1 datablock
//anz_page <=15 ---> ANZP ---> AnzP (_DBxx. DBB107)
//anz_page >=16 ---> 0    ---> AnzP (_DBxx. DBB107)
      A     DIX 460.0;	// Prüfen ob sich die Pageanzahl oder Startpage
      A(;	// geändert hat.
      O(;
      L     DIW 448;
      L     DIW 462;
      <>I;
      );
      O(;
      L     DBB 206;
      L     DIW 446;
      <>I;
      );
      );
      R     DIX 492.1;	// Reset wenn Unterschied
      A     DIX 492.1;	// Berechnung durchgeführt
      JC    a1_0;
      AN    DIX 492.0;	// Erste Berechnung starten
      JC    a1_1;
      A     DIX 492.0;	// Auswertung der nachfolgenden Startadressen
      A(;
      L     DIW 490;	// ist immer die zweite Berechnung
      L     2;	// bei mehr als 32 Page
      ==I;
      );
      JC    a1_2;	// Sprung bei 2 Loop's ---> bis 48 Page
      A     DIX 492.0;
      A(;
      L     DIW 490;	// ist immer die zweite Berechnung
      L     1;	// bei mehr als 16 Page
      ==I;
      );
      JC    a1_3;	// Sprung bei 1 Loop's ---> bis 32 Page
      JU    a1_0;	// keine weitere Berechnung durchführen
//-------------------ermittlung Startpage-------------------
a1_1: S     DIX 492.1;	// bis 16 Page
      L     DIW 448;
      T     DIW 462;
      L     DIW 446;
      T     DBB 206;	// Startpage setzten
      L     DIW 448;
      L     16;
      >I;
      JC    a1_6;	// mehr als 16 Page
      L     DIW 448;
      JU    a1_4;	// weniger als 16 Page
//----------------------------------------------------------
a1_6: L     DIW 448;	// Berechnung der 
      L     16;	// verbleibenden
      -I;	// Anzahl von Page's
      T     DIW 498;	// Restpage sichern
      L     16;	// es wird fest 16 geladen
      JU    a1_4;	// da es noch mehr als 16 Page sind
//----------------------------------------------------------
a1_2: S     DIX 492.1;	// mehr als 32 Page
      L     DBB 206;
      L     16;
      +I;
      T     DBB 206;	// neue Startpage setzten
      L     DIW 498;
      L     16;
      >I;
      JC    a1_5;	// mehr als 16 Page
      L     DIW 498;
      JU    a1_4;
//-----------------------------------------------------------
a1_5: L     DIW 498;	// siehe a1_6
      L     16;
      -I;
      T     DIW 498;
      L     16;
      JU    a1_4;
//-----------------------------------------------------------
a1_3: S     DIX 492.1;	// mehr als 16 Page
      L     DBB 206;
      L     16;
      +I;
      T     DBB 206;	// neue Startpage setzten
      L     DIW 498;
//-----------------------------------------------------------
a1_4: T     DIW 464;	// Anzahl Page ermitteln
//-----------------------------------------------------------
a1_0: L     DIW 464;	// Anzahl Page laden
      L     16;
      <I;
      JC    a1_7;	// bei mehr als 16 Page
      L     0;	// wird Null geladen (vom System vorgegeben)
      JU    a1_8;	// und eingetragen
//-----------------------------------------------------------
a1_7: TAK;	// bei weniger als 16 Page, 
//                                        wird die reale Menge geladen
//-----------------------------------------------------------
a1_8: T     DBB 207;	// Anzahl Page eintragen
NETWORK
TITLE = Ermittelung der Schleifenanzahl
//wird benötigt wenn mehr als 16 Page gelesen oder geschrieben werden sollen.
//
//----------------------- Loop ermittel----------------------
      L     DIW 448;
      L     16;
      <=I;
      JC    b1_4;
      O     DIX 492.0;
      ON    DIX 460.5;
      JC    b1_6;
      L     DIW 448;
      L     32;
      >I;
      JC    b1_2;
      L     DIW 448;
      L     16;
      >I;
      JC    b1_3;
      JU    b1_4;
b1_2: L     3;	// Wert 3 wenn ANZP >32
      S     DIX 492.0;
      JU    b1_5;
b1_3: L     2;	// Wert 2 wenn ANZP >16
      S     DIX 492.0;
      JU    b1_5;
b1_4: R     DIX 492.0;	// Wert 0 wenn ANZP <=16
      L     0;
b1_5: T     DIW 490;
b1_6: NOP   0;
NETWORK
TITLE = Read steuerblock (8 bytes) und transferiere in den _DB 
//Es wird geprüft ob der E/A-Bereich oder der Peripheriebereich konfiguriert ist 
//danach werden die Daten von den Eingängen gelesen und in den _DB übertragen.
//Die 8 Bytes sind die Rückmeldungen vom OIS-L.
      L     DIW 450;
      L     1;
      ==I;
      JC    c1_1;
      L     P#0.0;
      L     DIW 452;
      SLD   3;
      +D;
      LAR1;
      L     ID [AR1,P#0.0];
      T     DBD 0;
      L     ID [AR1,P#4.0];
      T     DBD 4;
      JU    c1_0;
//------------------ Peripheriebereich------------------
c1_1: L     P#0.0;
      L     DIW 452;
      SLD   3;
      +D;
      LAR1;
      L     PID [AR1,P#0.0];
      T     DBD 0;
      L     PID [AR1,P#4.0];
      T     DBD 4;
c1_0: NOP   0;
NETWORK
TITLE = Überprüfe Datenlänge und CTL  Byte
      L     DBB 6;
      L     0;
      ==I;
      AN    DBX 7.0;
      A     DBX 7.2;
      =     DIX 493.4;
NETWORK
TITLE = Überprüfe Statusbyte auf Fehler
//Hier wird das Statusbyte eingelesen, auf Fehler geprüft und an den Ausgang 
//HW_FTL gelegt.
      L     DBB 2;
      T     DIB 458;
      L     B#16#F0;
      ==I;
      =     DIX 460.4;
NETWORK
TITLE = Lade controllbyte und transferiere zum State_HS 
//Hier wird das Controllbyte eingelesen und an den Ausgang 
//State_HS gelegt.
      L     DBB 7;
      T     DIB 459;
NETWORK
TITLE = Transfer ADB und DBN in _dB beim lesen
//Nur relevant beim Lesen. Anz Block und aktual Block eintragen.
      A(;
      A     DIX 442.2;
      JNB   _00b;
      L     1;
      T     DBB 208;
      SET;
      SAVE;
      CLR;
_00b: A     BR;
      );
      JNB   _013;
      L     DBB 208;
      T     DBB 209;
_013: NOP   0;
NETWORK
TITLE = Read: Datenlänge auf Null setzten
//Beim Lesen wird die Datenlänge fest auf Null gelegt.
      A     DIX 442.2;
      JNB   _014;
      L     0;
      T     DBB 210;
_014: NOP   0;
NETWORK
TITLE = Toggelbit neue Daten vom Slave vorhanden
//CTL Byte CTL.#1
//neue Daten vom slave vorhanden
      A(;
      O(;
      A     DBX 7.1;
      BLD   100;
      FP    DIX 492.3;
      );
      O(;
      A     DBX 7.1;
      BLD   100;
      FN    DIX 492.4;
      );
      );
      =     DIX 492.5;
      A     DIX 492.5;
      =     DIX 494.1;
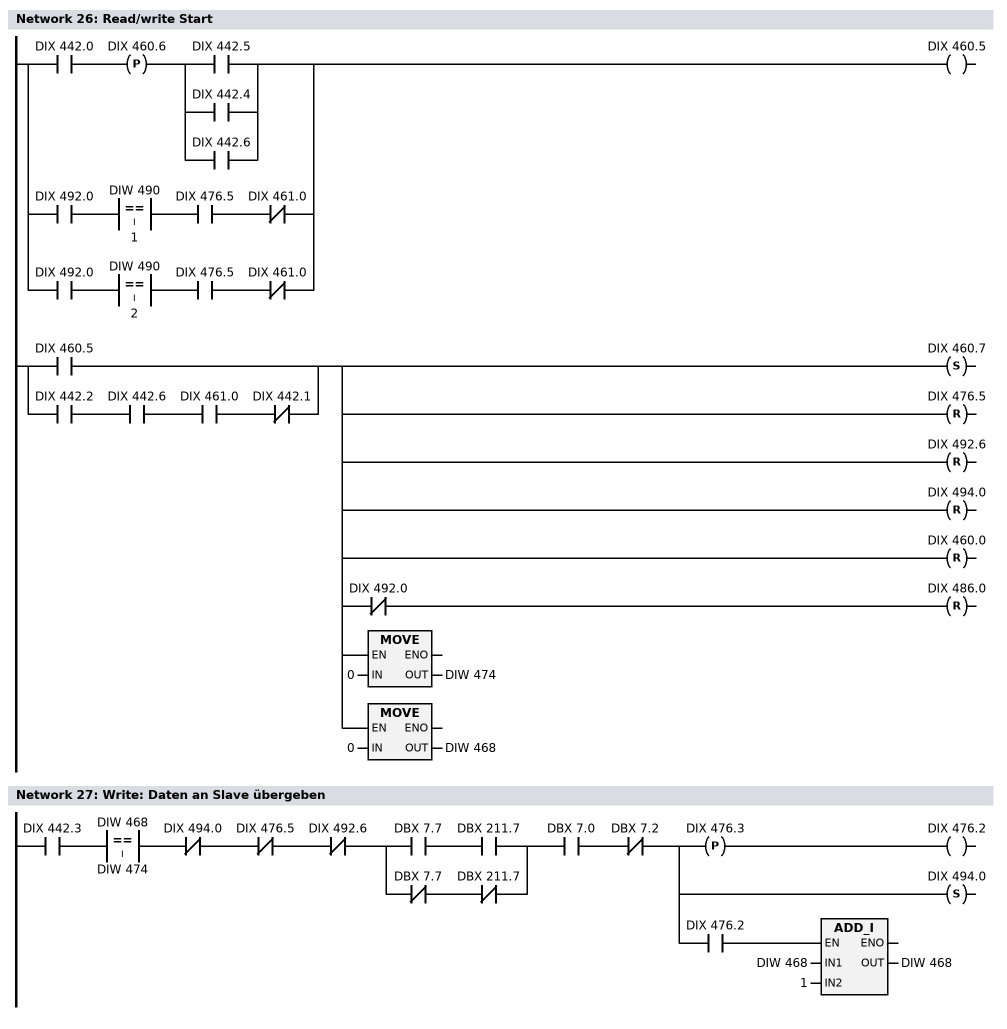
NETWORK
TITLE = Read/write Start
//Startflanke für Lesen und Schreiben setzten.
//Über die beiden Vergleicher wird geprüft ob noch mehr Daten gelesen oder 
//geschrieben werden sollen und ein neuer Transfer angestoßen.Im Cont-Modus muß 
//als start auch der Eingang Start_RW gesetzt werden.
      A(;
      A(;
      A     DIX 442.0;	//Convert into pointerformat
      BLD   100;
      FP    DIX 460.6;	//Write address into adressreg.1
      );	//Load input - 1st page 
      A(;
      O     DIX 442.5;	//Load input - 2nd page 
      O     DIX 442.4;
      O     DIX 442.6;
      );
      O;
      A     DIX 492.0;
      A(;
      L     DIW 490;
      L     1;
      ==I;
      );
      A     DIX 476.5;
      AN    DIX 461.0;
      O;
      A     DIX 492.0;
      A(;
      L     DIW 490;
      L     2;
      ==I;
      );
      A     DIX 476.5;
      AN    DIX 461.0;
      );
      =     DIX 460.5;
      A     DIX 460.5;
      O;
      A     DIX 442.2;
      A     DIX 442.6;
      A     DIX 461.0;
      AN    DIX 442.1;
      =     L 4.0;
      A     L 4.0;
      BLD   102;
      S     DIX 460.7;
      A     L 4.0;
      BLD   102;
      R     DIX 476.5;
      A     L 4.0;
      BLD   102;
      R     DIX 492.6;
      A     L 4.0;
      BLD   102;
      R     DIX 494.0;
      A     L 4.0;
      BLD   102;
      R     DIX 460.0;
      A     L 4.0;
      AN    DIX 492.0;
      R     DIX 486.0;
      A     L 4.0;
      JNB   _015;
      L     0;
      T     DIW 474;
_015: NOP   0;
      A     L 4.0;
      JNB   _016;
      L     0;
      T     DIW 468;
_016: NOP   0;
NETWORK
TITLE = Write: Daten an Slave übergeben 
//DBX7.0 Daten gültig
//DBX7.2 Aufrag läuft
//DBX7.7 = DBX211.7 Slave quittiert neue Daten emfangen
      A     DIX 442.3;
      A(;
      L     DIW 468;
      L     DIW 474;
      ==I;
      );
      AN    DIX 494.0;
      AN    DIX 476.5;
      AN    DIX 492.6;
      A(;
      A     DBX 7.7;
      A     DBX 211.7;
      O;
      AN    DBX 7.7;
      AN    DBX 211.7;
      );
      A     DBX 7.0;
      AN    DBX 7.2;
      =     L 4.0;
      A     L 4.0;
      FP    DIX 476.3;
      =     DIX 476.2;
      A     L 4.0;
      BLD   102;
      S     DIX 494.0;
      A     L 4.0;
      A     DIX 476.2;
      JNB   _017;
      L     DIW 468;
      L     1;
      +I;
      T     DIW 468;
_017: NOP   0;
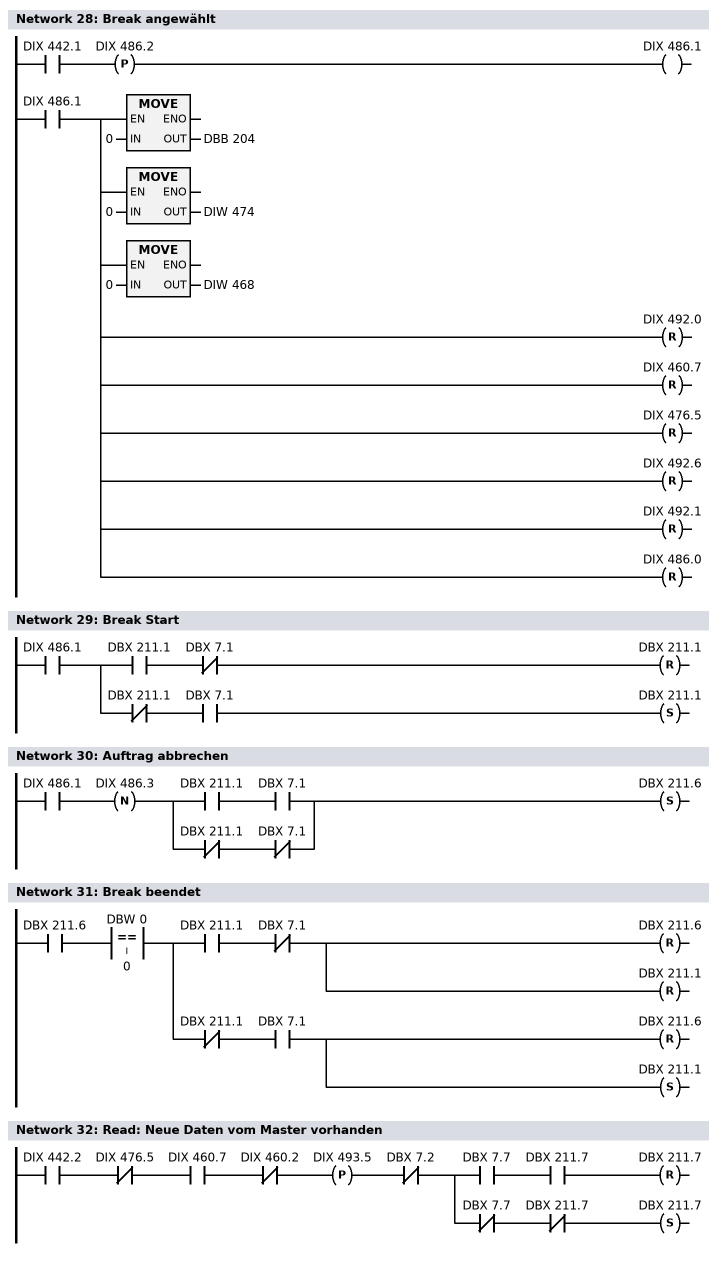
NETWORK
TITLE = Break angewählt
//Start Break: Rücksetzten und löschen aller relevanter Daten
      A(;
      A     DIX 442.1;
      BLD   100;
      FP    DIX 486.2;
      );
      =     DIX 486.1;
      A     DIX 486.1;
      =     L 4.0;
      A     L 4.0;
      JNB   _01b;
      L     0;
      T     DBB 204;
_01b: NOP   0;
      A     L 4.0;
      JNB   _01d;
      L     0;
      T     DIW 474;
_01d: NOP   0;
      A     L 4.0;
      JNB   _01e;
      L     0;
      T     DIW 468;
_01e: NOP   0;
      A     L 4.0;
      BLD   102;
      R     DIX 492.0;
      A     L 4.0;
      BLD   102;
      R     DIX 460.7;
      A     L 4.0;
      BLD   102;
      R     DIX 476.5;
      A     L 4.0;
      BLD   102;
      R     DIX 492.6;
      A     L 4.0;
      BLD   102;
      R     DIX 492.1;
      A     L 4.0;
      BLD   102;
      R     DIX 486.0;
NETWORK
TITLE = Break Start
//CTL.1(Out)=CTL.1(In)
      A     DIX 486.1;
      =     L 4.0;
      A     L 4.0;
      A     DBX 211.1;
      AN    DBX 7.1;
      R     DBX 211.1;
      A     L 4.0;
      AN    DBX 211.1;
      A     DBX 7.1;
      S     DBX 211.1;
NETWORK
TITLE = Auftrag abbrechen
//CTL.6(Out)=1 wird gesetzt.Break Befehl für den OIS-L Kontroller eingeleitet.
      A     DIX 486.1;
      FN    DIX 486.3;
      A(;
      A     DBX 211.1;
      A     DBX 7.1;
      O;
      AN    DBX 211.1;
      AN    DBX 7.1;
      );
      S     DBX 211.6;
NETWORK
TITLE = Break beendet
//CTL.6=0 setzten
//CTL.1(out)=CTL.1(In)
//Abfrage des KDO, wenn Null und DBX7.1 hat quittiert, dann wird der Break-Befehl
//zurückgesetzt. Break durchgeführt!
      A     DBX 211.6;
      A(;
      L     DBW 0;
      L     0;
      ==I;
      );
      =     L 4.0;
      A     L 4.0;
      A     DBX 211.1;
      AN    DBX 7.1;
      R     DBX 211.6;
      R     DBX 211.1;
      A     L 4.0;
      AN    DBX 211.1;
      A     DBX 7.1;
      R     DBX 211.6;
      S     DBX 211.1;
NETWORK
TITLE = Read: Neue Daten vom Master vorhanden
//CTL.7 toggeln, CTL.7 zeigt dem Slave die neue Komandobeauftragung an.
      A     DIX 442.2;
      AN    DIX 476.5;
      A     DIX 460.7;
      AN    DIX 460.2;
      FP    DIX 493.5;
      AN    DBX 7.2;
      =     L 4.0;
      A     L 4.0;
      A     DBX 7.7;
      A     DBX 211.7;
      R     DBX 211.7;
      A     L 4.0;
      AN    DBX 7.7;
      AN    DBX 211.7;
      S     DBX 211.7;
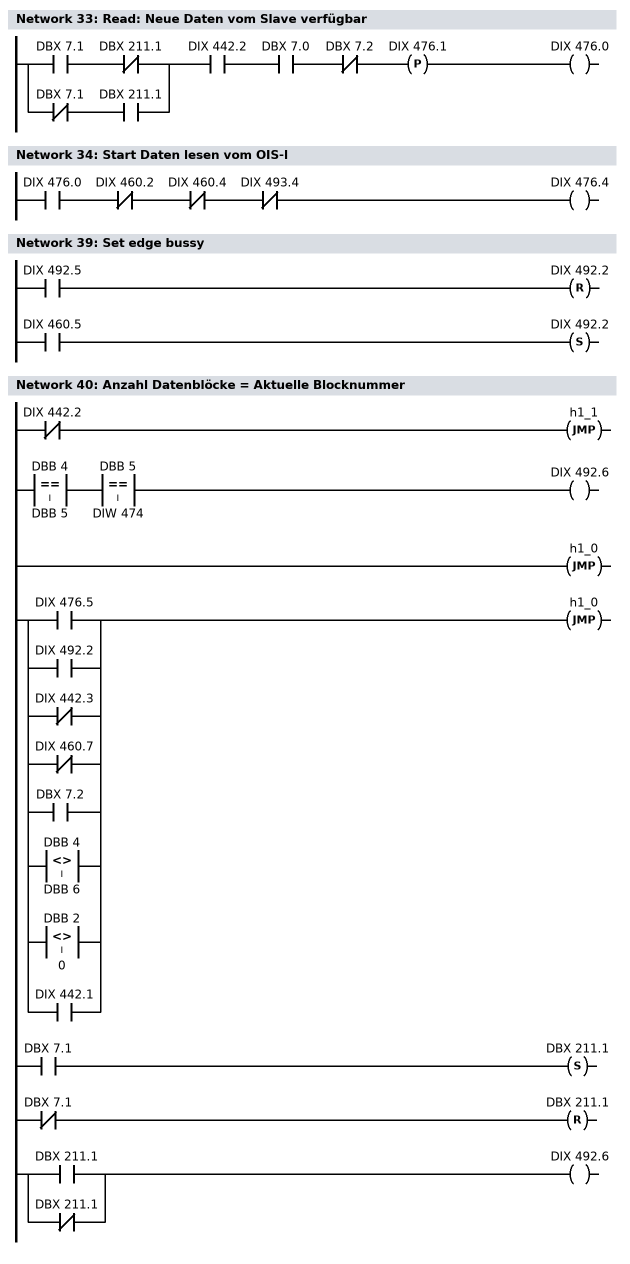
NETWORK
TITLE = Read: Neue Daten vom Slave verfügbar
//Das CTL.1(in) signalisiert neue Daten.
      A(;
      A     DBX 7.1;
      AN    DBX 211.1;
      O;
      AN    DBX 7.1;
      A     DBX 211.1;
      );
      A     DIX 442.2;
      A     DBX 7.0;
      AN    DBX 7.2;
      FP    DIX 476.1;
      =     DIX 476.0;
NETWORK
TITLE = Start Daten lesen vom OIS-l
//RD startet das einlesen der daten von den Eingängen.
      A     DIX 476.0;	//No read mode
      AN    DIX 460.2;	//No new data block
      AN    DIX 460.4;
      AN    DIX 493.4;	//End of reading
      =     DIX 476.4;
NETWORK
TITLE = Berechnung Anzahl Byte's und Anzahl Blocks
//anz_bytes=ANZP*4
//Anz_blocks=anz_byts/24
//Rest im akku1 H
//wenn rest => inc1<akku1>
      A     DIX 460.7;
      JC    d1_0;
      L     DW#16#0;	// Akku auf Null setzten
      L     DIW 464;	// Anzahl Bytes berechnen
      L     4;
      *I;
      T     DIW 472;	// speichern in anz_bytes
      T     DIW 470;	// und rest_bytes
      L     24;	// Anzahl Blocks berechnen
      /I;
      T     DIW 466;	// Anzahl Blocks sichern
      SRD   16;	// <akku1-h> ---> in den akku1-l schieben
      L     0;	// Überprüfung ob Rest vorhanden
      ==I;
      JC    d1_1;	// wenn <akku1> = 0 kein Rest
      L     DIW 466;	// wenn <akku1> <> 0 erhöhe die Blockzahl um eins
      INC   1;	// wenn Rest dann Blockanzahl +1
      T     DIW 466;
d1_1: AN    DIX 442.3;	// im Schreibmodus wird die Blockanzahl
      JC    d1_0;
      L     DIW 466;	// an den OIS-L Kontroller gesandt
      T     DBB 208;
d1_0: NOP   0;
NETWORK
TITLE = Berechnung der Startadresse für den Pointer (Lesen)
//((Startpage-16)*4)+8=Pointer_buffer
//
//16  --> min. Startpage
//4   --> Byte pro Page
//8 --> Startadresse im _DB (Datenbereich lesen)
      O     DIX 486.0;
      ON    DIX 442.2;
      O     DIX 442.1;
      JC    e1_0;
      L     0;
      L     DIW 446;
      <>I;
      JC    e1_1;	// nach jedem Start_RD wird der Pointer
      JU    e1_2;
e1_1: L     16;	// nach obriger Formel neu berechnet
      -I;
e1_2: T     DID 478;
      L     4;
      *I;
      T     DID 478;
      L     P#8.0;
      L     DID 478;
      SLD   3;
      +D;
      T     DID 482;
      S     DIX 486.0;	// Verriegelung Pointer ist berechnet
e1_0: NOP   0;
NETWORK
TITLE = Berechnung Loop_Counter
//Für das Lesen und Schreiben werden hier die Schleifendurchlaüfe berechnet.
//Für eine Page muß die Schleife 1 mal durchlaufen werden. 1Page = 4 Bytes 
      L     DIW 474;
      L     0;
      >I;
      JC    f1_1;	// mehr als 1 Block ?
      L     DIW 464;
      L     6;
      >I;
      JC    f1_1;	// Pageanzahl >6
      TAK;	// Anzahl Page in den Akku 1 laden
      JU    f1_0;	// und zum Ende springen
f1_1: L     DIW 474;
      L     0;
      >I;
      JC    f1_2;	// mehr als 1 Block ?
      L     6;
      JU    f1_0;
f1_2: A     DIX 442.3;
      JC    f1_3;	// Modus Schreiben springe --> f1_3 
      L     DBB 6;	// Modus Lesen: aktuelle Datenlänge laden
      L     4;
      /I;	// und durch 4 teilen
      JU    f1_0;	// zum Ende springen
f1_3: L     DIW 470;	// Modus Schreiben: errechnete Restbytes laden
      L     24;	// und vergleichen ob mehr als 24 Byts
      >=I;	// noch geschrieben werden müssen
      JC    f1_4;	// wenn >24 springe ---> f1_4
      TAK;	// wenn < 24: alten Akkuinhalt zurückholen
f1_4: L     4;
      /I;	// teilen und 
f1_0: T     DIW 488;	// Eintrag anz_loop
NETWORK
TITLE = Read: Store data
      ON    DIX 442.2;
      ON    DIX 476.4;
      O     DIX 442.1;
      JC    g1_0;
      L     P#8.0;	// Pointer Adressraum Setzten
      L     DIW 452;
      SLD   3;
      +D;
      T     DID 500;
      L     DIW 488;	// Anzahl Loop's laden
//----------------Start Einleseroutine---(Loop-Routine)--------
g1_2: T     DIW 508;
      L     DIW 450;	// E/A-Bereich oder Peripheriebereich
      L     1;
      ==I;
      JC    g1_3;	// sprung wenn EA-or_PW = log. 1
//-------------------- EA-Bereich -------------------------
      L     DID 500;	// Pointer laden
      LAR1;
      L     ID [AR1,P#0.0];	// Zeiger auf Eingänge
      L     DID 482;
      LAR1;	// Daten laden
      TAK;
      T     DBD [AR1,P#0.0];	// und im Datenbereich _DB ablegen
      JU    g1_4;	// sprung ---> Pointer erhöhen
//-------------------- Peripheriebereich ------------------
g1_3: L     DID 500;	// siehe EA-Bereich
      LAR1;
      L     PID [AR1,P#0.0];
      L     DID 482;
      LAR1;
      TAK;
      T     DBD [AR1,P#0.0];
//-------------------- Pointer erhöhen --------------------
g1_4: L     DID 500;	// Pointer_Input und 
      L     P#4.0;
      +D;
      T     DID 500;
      L     DID 482;	// Pointer_buffer
      L     P#4.0;	// werden um 4 erhöht
      +D;
      T     DID 482;
      L     DIW 508;	// loop_counter laden und
      LOOP  g1_2;	// decrementieren bis 0 erreicht ist
// ------------------- Controllbits toggel ----------------
      A     DBX 7.1;	// CTL.1(out) toggeln
      S     DBX 211.1;	// CLT.1(in) = CLT.1(out)
      AN    DBX 7.1;
      R     DBX 211.1;
      L     DIW 474;	// Anzahl gelesener
      L     1;	// Blöcke erhöhen
      +I;
      T     DIW 474;	// und in rcv_blocks speichern 
g1_0: NOP   0;
NETWORK
TITLE = Set edge bussy
      A     DIX 492.5;
      R     DIX 492.2;
      A     DIX 460.5;
      S     DIX 492.2;
      NOP   0;
NETWORK
TITLE = Anzahl Datenblöcke = Aktuelle Blocknummer
//Quittierungssignal beim lesen/schreiben wenn die Daten komplett 
//gelesen/geschrieben und abgespeichert sind.
//----------------------Lesen-------------------------------
      ON    DIX 442.2;
      JC    h1_1;	// wenn nicht Lesen dann zum UP h1_1
      A(;
      L     DBB 4;
      L     DBB 5;
      ==I;
      );
      A(;
      L     DBB 5;
      L     DIW 474;
      ==I;
      );
      =     DIX 492.6;
      JU    h1_0;
//-----------------------Schreiben---------------------------
h1_1: NOP   0;
      O     DIX 476.5;
      O     DIX 492.2;
      ON    DIX 442.3;
      ON    DIX 460.7;
      O     DBX 7.2;
      O(;
      L     DBB 4;
      L     DBB 6;
      <>I;
      );
      O(;
      L     DBB 2;
      L     0;
      <>I;
      );
      O     DIX 442.1;
      JC    h1_0;
//---------------------CTL.1 toggeln--------------------------
      A     DBX 7.1;
      S     DBX 211.1;
      AN    DBX 7.1;
      R     DBX 211.1;
      O     DBX 211.1;
      ON    DBX 211.1;
      =     DIX 492.6;	// CTL.1 getoggelt Auftrag Ende Merker
h1_0: NOP   0;
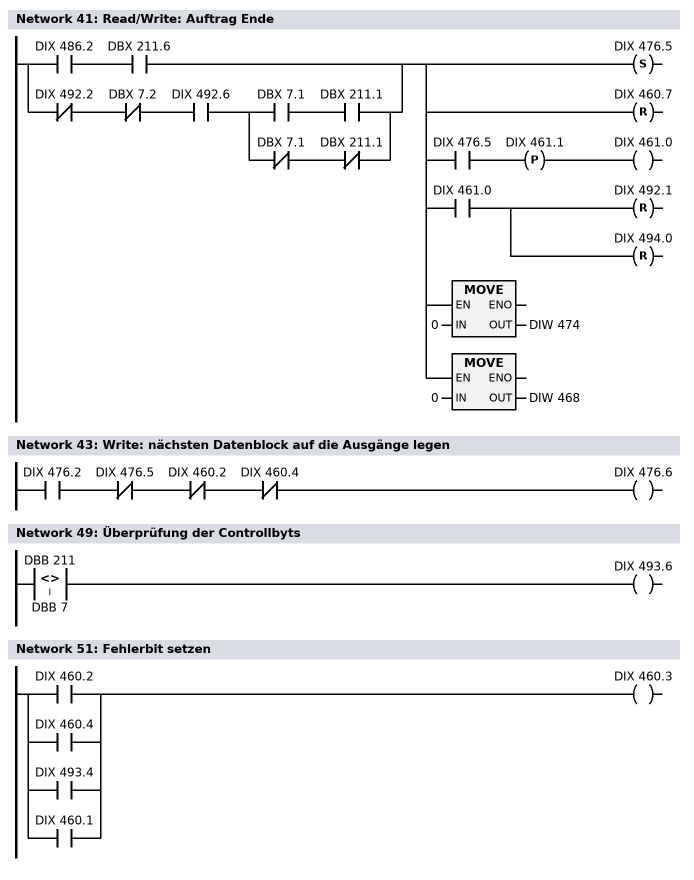
NETWORK
TITLE = Read/Write: Auftrag Ende 
      A     DIX 486.2;
      A     DBX 211.6;
      O;
      AN    DIX 492.2;
      AN    DBX 7.2;
      A     DIX 492.6;
      A(;
      A     DBX 7.1;
      A     DBX 211.1;
      O;
      AN    DBX 7.1;
      AN    DBX 211.1;
      );
      =     L 4.0;
      A     L 4.0;
      BLD   102;
      S     DIX 476.5;
      A     L 4.0;
      BLD   102;
      R     DIX 460.7;
      A     L 4.0;
      A     DIX 476.5;
      FP    DIX 461.1;
      =     DIX 461.0;
      A     L 4.0;
      A     DIX 461.0;
      R     DIX 492.1;
      R     DIX 494.0;
      A     L 4.0;
      JNB   _01f;
      L     0;
      T     DIW 474;
_01f: NOP   0;
      A     L 4.0;
      JNB   _021;
      L     0;
      T     DIW 468;
_021: NOP   0;
NETWORK
TITLE = Loop Counter für mehrfach lesen decrementieren
//Der Loop Counter dient dazu, bei mehr als 16 Page den Lese oder Schreibvorgang 
//erneut zu starten. Im cont Mode ist ein lesen von mehr als 16 Page nicht 
//möglich.
      ON    DIX 461.0;
      ON    DIX 492.0;
      JC    i1_0;
      L     DIW 490;
      DEC   1;
      T     DIW 490;
      L     0;
      ==I;
      A     DIX 492.0;
      R     DIX 492.0;
i1_0: A     DIX 476.5;
      AN    DIX 460.0;
      A(;
      L     DIW 490;
      L     0;
      ==I;
      );
      S     DIX 460.0;	//Auftrag abgearbeitet
NETWORK
TITLE = Write: nächsten Datenblock auf die Ausgänge legen
      A     DIX 476.2;	//and no condition write next block
      AN    DIX 476.5;
      AN    DIX 460.2;
      AN    DIX 460.4;	//or Break
      =     DIX 476.6;
NETWORK
TITLE = Datenübergabe zum OIS-L kann gestartet werden
//aktiv im Modus Write
      ON    DIX 493.7;	// Daten auf die Ausgänge gelegt: Log 1
      JC    z1_0;	// noch keine Daten auf den Ausgängen: Log 0
//-------------------------CTL.7 (out) toggeln-------------------
      AN    DIX 476.5;
      A     DBX 7.7;
      R     DBX 211.7;
      AN    DIX 476.5;
      AN    DBX 7.7;
      S     DBX 211.7;
//------------------------Blockanzahl erhöhen und Dlen bestimmen-------- 
      L     DIW 474;
      L     1;
      +I;
      T     DIW 474;
      T     DBB 209;	// aktuellen Block eintragen
      L     DIW 470;
      L     24;
      >=I;
      JC    z1_1;
      TAK;
z1_1: T     DBB 210;	// aktuelle Datenlänge eintragen
      L     DIW 470;
      L     DBB 210;	// Restdatenlänge bestimmen
      -I;
      T     DIW 470;
      R     DIX 494.0;
      R     DIX 493.7;
      L     DIW 470;
      L     0;
      ==I;
      S     DIX 494.0;
z1_0: NOP   0;
NETWORK
TITLE = Berechnung der Startadresse für den Pointer (Schreiben)
//((Startpage-16)*4)+212= RD_Pointer_dest
//
//16  --> min. Startpage
//4   --> Byte pro Page
//212 --> Startadresse im _DB (Datenbereich schreiben)
      O     DIX 486.0;
      ON    DIX 442.3;
      O     DIX 442.1;
      JC    j1_0;
//-----------------------------------------------------
      L     DIW 446;
      L     16;
      -I;
      T     DID 478;
      L     4;
      *I;
      T     DID 478;
      L     P#212.0;
      L     DID 478;
      SLD   3;
      +D;
      T     DID 482;
      S     DIX 486.0;
j1_0: NOP   0;
NETWORK
TITLE = Setze Startadresse Ausgänge
      L     P#8.0;	//  Anfangsadresse des Adressbereichs für die Daten
      L     DIW 454;
      SLD   3;	// Umwandlung ins Pointerformat
      +D;
      T     DID 504;	// Pointeradresse setzten
NETWORK
TITLE = Write: Data to OIS
      ON    DIX 442.3;
      ON    DIX 476.6;
      O     DIX 442.1;
      JC    L1_0;
      L     DIW 488;
//-----------------Schleife für Datenübergabe------------
L1_1: T     DIW 508;	// Schleife Datenübergabe start
      L     DIW 450;	// Auswertung E/A oder Peripheriebereich
      L     1;
      ==I;
      JC    L1_2;
//------------------ EA-Bereich -------------------------
      L     DID 482;	// Datenbereich pointer laden
      LAR1;
      TAK;
      L     DBD [AR1,P#0.0];	// Daten aus _DB holen
      L     DID 504;	// Ausgangspointer laden
      LAR1;
      TAK;
      T     QD [AR1,P#0.0];	// Daten auf Ausgänge schreiben
      JU    L1_3;
//------------------ Perihperiebereich ------------------
L1_2: L     DID 482;	// siehe EA-Bereich
      LAR1;
      TAK;
      L     DBD [AR1,P#0.0];
      L     DID 504;
      LAR1;
      TAK;
      T     PQD [AR1,P#0.0];
//------------------ Pointer erhöhen --------------------
L1_3: L     DID 482;
      L     P#4.0;
      +D;
      T     DID 482;
      L     DID 504;
      L     P#4.0;
      +D;
      T     DID 504;
      L     DIW 508;
      LOOP  L1_1;	// Schleife Datenübergabe ende
//------------------ Daten OK ---------------
      S     DIX 493.7;
L1_0: NOP   0;
NETWORK
TITLE = Read/write: Transfer commandoblock
      L     DIW 450;
      L     1;
      ==I;
      JC    m1_1;
//------------------ EA-Bereich -------------------------
      L     P#0.0;
      L     DIW 454;
      SLD   3;
      +D;
      LAR1;
      L     DBD 204;
      T     QD [AR1,P#0.0];
      L     DBD 208;
      T     QD [AR1,P#4.0];
      JU    m1_0;
//------------------ Perihperiebereich ------------------
m1_1: L     P#0.0;
      L     DIW 454;
      SLD   3;
      +D;
      LAR1;
      L     DBD 204;
      T     PQD [AR1,P#0.0];
      L     DBD 208;
      T     PQD [AR1,P#4.0];
m1_0: NOP   0;
NETWORK
TITLE = Überprüfung der Controllbyts
//Ist DBB 211 <> DBB7 dann starte Timeout
      L     DBB 211;
      L     DBB 7;
      <>I;
      =     DIX 493.6;
NETWORK
TITLE = [1.0] Timeout 
//Baumer: S5 Timer(T_OUT) replace with counter #BUZ_OutTimeOut
      A     DIX 493.6;
      JC    TOJ1;
      L     DIW 456;
      T     DIW 422;
      JU    TOJ2;
TOJ1: L     0;
      L     DIW 422;
      >=I;
      ON    "GCS7_Gr_OutTick200ms";
      JC    TOJ2;
      L     200;
      -I;
      T     DIW 422;
TOJ2: L     0;
      <=I;
      O;
      A     DIX 460.1;
      AN    DIX 476.5;
      =     DIX 460.1;
NETWORK
TITLE = Fehlerbit setzen
Out:  O     DIX 460.2;
      O     DIX 460.4;
      O     DIX 493.4;
      O     DIX 460.1;
      =     DIX 460.3;
NETWORK
TITLE = [1.0] BUZ: Command from Buhler to Baumer RFID (Part 2)
// (network holds code this reader does not know; not shown)
//-Reader idling---
// 
// 
//-Reset commands---
// 
// 
//-Reading done---
// 
// 
//-Fault handling---
//WinTrend      U     #ToBuhler.RFIDJobRunning
//WinTrend      L     S5T#150MS
//WinTrend      SV    T    202
//WinTrend      U     T    202
//WinTrend      =     M   1400.2
// 
// 
//WinTrend      L     S5T#150MS
//WinTrend      SV    T    201
//WinTrend      U     T    201
//WinTrend      =     M   1400.1
NETWORK
TITLE = [1.0] BUZ: Retry Counter
      A     DIX 410.0;
      AN    DIX 410.2;
      JC    BRJ1;
      R     DIX 410.2;
      L     0;
      T     DIW 430;
      JU    BRJ2;
BRJ1: L     DIW 430;
      A     DIX 442.1;
      FP    DIX 420.4;
      JCN   BRJ2;
      +     1;
      T     DIW 430;
BRJ2: L     5;
      >=I;
      =     DIX 420.0;
      R     DIX 420.3;
END_FUNCTION_BLOCK

FUNCTION "SYS_CBitCtrl" : VOID	// FC 2
TITLE = Change bit controller
//COPYRIGHT:   (C) 1994 BY  BUHLER LTD
//                          CH-9240 UZWIL  SWITZERLAND
//
//PRODUCT:     GCS7
//
//TITLE:       FC 002 METHOD'S FOR      CHANGE-BIT-DB
//                    METHODEN FUER AENDERUNGS-BIT-DB
//
//-------------------------------------------------------------------------
//
//IDENT:       AUTOR:              DEPT:                           DATE:
//
//FC2.1.1      A.Egli              CT3                             08-Nov-20002
//             New release
//FC002.1B     A.Egli              CT3                             2-Dec-99
//             RELEASE 1A Convert form S5
//FC002.1A     A.Egli               AEE61                          11-Nov-96
//             RELEASE 1A Convert form S5
//
//-------------------------------------------------------------------------
//
//-------------------------------------------------------------------------
//
//PURPOSE:     MANUAL : ....... .DOC
//             
//
//RESTRICTIONS:
//
//-------------------------------------------------------------------------
//
//
//COPYRIGHT:          (C) 1990 BY  BUHLER LTD
//                                 CH-9240 UZWIL  SWITZERLAND
//
//PRODUCT:            GCS7
//
//TITLE:              FC 002 METHOD'S FOR      CHANGE-BIT-DB
//                           METHODEN FUER AENDERUNGS-BIT-DB
//
//-------------------------------------------------------------------------
//
//IDENT:              SSW.FC002.1B     A.Egli   CT3              2-Dec-99
//                       RELEASE 1A Convert form S5
//IDENT:              SSW.FC002.1A     A.Egli   AEE61           11-Nov-96
//                       RELEASE 1A Convert form S5
//
//-------------------------------------------------------------------------
//
//PURPOSE:            MANUAL : CBIT1MAN.DOC
//                   
//
//RESTRICTIONS:       ACCU1 =Code
//
//-------------------------------------------------------------------------
//
//
AUTHOR : EA
FAMILY : GCS7SYS
NAME : MET_CBIT
VERSION : 1.1
VAR_TEMP
  tmpCBit : ARRAY  [1 .. 4 ] OF //Must by at LB0
  BOOL ;
  CODE : INT ;	//Function code of the to compute function
  tmpAddrPointer : DINT ;
  tmpAddrCopyBit : DINT ;
  tmpDBSource : INT ;
  tmpDWSource : DINT ;
  tmpAddrEnd : DINT ;
  tmpCBitOld : DWORD ;
  tmpFcClear : BOOL ;
  tmpBitNr : INT ;
END_VAR
BEGIN
NETWORK
TITLE =
      T     #CODE;
NETWORK
TITLE = CBit: Code=3
//Set Changebit of GCS90 objects:
//
//Input  : AR2        : Address dynamic data
//         DB2.DBW12  : ParBlockLen
//Output : F13.0 /F13.1 /F13.2 /F13.3
//
      L     #CODE;
      L     3;
      <>I;
      JC    F1;
      TAR2;
      L     "SYS_CBitDB".ParBlockLen;	//ParBlockLen (Byte)
      SLD   3;	//Length in Bit
      /I;
      T     #tmpBitNr;
      L     3;
      >=I;
      JC    BIT4;
      L     #tmpBitNr;
      L     1;
      SLW;
      L     "GCS7_Gr_ElMaToGroup2";	//Changebit.CBIT[1..4] 
      OW;
      T     "GCS7_Gr_ElMaToGroup2";	//-->Changebit.CBIT[1..4] 
//---Blockgrenze---
      TAR2;
      +     L#48;
      L     "SYS_CBitDB".ParBlockLen;	//ParBlockLen (Byte)
      SLD   3;	//Length in Bit
      /I;
      T     #tmpBitNr;
      L     3;
      >=I;
      JC    BIT4;
      L     #tmpBitNr;
      L     1;
      SLW;
      L     "GCS7_Gr_ElMaToGroup2";	//Changebit.CBIT[1..4] 
      OW;
      T     "GCS7_Gr_ElMaToGroup2";	//-->Changebit.CBIT[1..4] 
      BEU;
BIT4: S     "GCS7_Gr_InCBit4";	//Changebit.CBit4
      BEU;
NETWORK
TITLE =  Read/copy
//Copy change bits from object DB to change bit DB to area 'Copy[x]' 
//
F1:   L     #CODE;
      L     1;
      <>I;
      JC    bEnd;
      R     #tmpFcClear;	// 2nd Loop for clear 
Clr:  OPN   "SYS_CBitDB";	// >>> call FIRST CBIT-DB
// Begin Loop 1: CBit-DB ---  
ZYK1: L     DBLG;
      +     -4;
      SLD   3;
      T     #tmpAddrEnd;
      L     DBW 10;	//  ParDWCopyByts
      SLD   3;
      LAR1;	//  -->tmpAddrCopyBit; 
      L     P#160.0;
      +D;
      T     #tmpAddrPointer;
// Begin Loop 2:Copy Change Bit -------- 
BEG2: L     DBD [#tmpAddrPointer];	// Pointer to Source address
      L     W#16#FFFF;
      AD;
      SLD   3;
      T     #tmpDWSource;
      L     DBW [#tmpAddrPointer];	// Pointer to Source address
      T     #tmpDBSource;
      L     -1;	// --> End of configuration
      L     #tmpDBSource;
      ==I;	//  
      JC    NEX1;	//  
      L     0;	//  
      ==I;	//  
      JC    NEX2;	//--> spare
      OPN   DI [#tmpDBSource];
      AN    #tmpFcClear;
      JC    Copy;
//--- Clear Change bit in object DB's 
      L     DIB [#tmpDWSource];
      L     2#11110000;	// Only 4 Bit per object  
      AW;
      T     DIB [#tmpDWSource];
      JU    NEX2;
//--- Copy Change bit ------- 
Copy: L     DIB [#tmpDWSource];
      L     2#1111;	// Only 4 Bit per object  
      AW;
      T     LB 0;	// tmpCBit     
      A     #tmpCBit[1];
      S     DBX [AR1,P#0.0];	// -->Copy[x]
      A     #tmpCBit[2];
      S     DBX [AR1,P#0.1];	// -->Copy[x+1]
      A     #tmpCBit[3];
      S     DBX [AR1,P#0.2];	// -->Copy[x+2]
      A     #tmpCBit[4];
      S     DBX [AR1,P#0.3];	// -->Copy[x+3]
NEX2: L     #tmpAddrPointer;
      +     32;
      T     #tmpAddrPointer;	// Pointer to next source DB        
      L     #tmpAddrEnd;
      >D;
      JC    NEX1;
      +AR1  P#0.4;	// Inc. address of copy bits
      JU    BEG2;
// End of Loop 2: -----
NEX1: L     0;	// 
      L     DBW 6;	// ParNextDB
      ==I;	// 
      JC    bOut;
      OPN   DB [DBW 6];	// Call Next DB 
      JU    ZYK1;
bOut: AN    #tmpFcClear;
      S     #tmpFcClear;
      JC    Clr;	//-->2nd Loop for clear 
      BEU;
bEnd: NOP   0;
NETWORK
TITLE =  FUNC=2, Update
//- Reset change bit CBit[x], if PC has accepted
//- Copy the Copy[x] to CBir[x]
//  
      L     #CODE;
      L     2;
      <>I;
      JC    dEnd;
      OPN   "SYS_CBitDB";
// Begin Loop 1:Copy Change Bit -------- 
dZY1: LAR1  P#0.0;
      L     DBW 10;	//ParDWCopyByts
      SLD   3;
      T     #tmpAddrCopyBit;
dZY2: L     DBD [AR1,P#40.0];	// RBit[x]
      INVD;
      L     DBD [AR1,P#200.0];	// CBit[x]
      AD;
      T     #tmpCBitOld;
      L     DBD [#tmpAddrCopyBit];
      OD;
      T     DBD [AR1,P#200.0];	// -->CBit[x]
      L     0;	// 
      T     DBD [AR1,P#40.0];	// -->RBit[x]
//   Increment address pointer  
      L     #tmpCBitOld;
      L     DBD [#tmpAddrCopyBit];
      AD;
      T     DBD [#tmpAddrCopyBit];
      L     #tmpAddrCopyBit;
      L     P#4.0;
      +D;
      T     #tmpAddrCopyBit;
      +AR1  P#4.0;
      TAR1;
      L     P#160.0;
      <D;
      JC    dZY2;
// End of Loop 2: -----
      L     0;	// 
      L     DBW 6;	// ParNextDB
      ==I;	// 
      BEC;
      OPN   DB [DBW 6];	// Call Next DB 
      JU    dZY1;	// 
dEnd: NOP   0;
NETWORK
TITLE =  END
END_FUNCTION

FUNCTION "SYS_DirectCtrl" : VOID	// FC 3
TITLE = PCControl
//COPYRIGHT:   (C) 1994 BY  BUHLER LTD
//                          CH-9240 UZWIL  SWITZERLAND
//
//PRODUCT:     GCS7
//
//TITLE:       FC3  Help Function Diagnositc interface
//
//-------------------------------------------------------------------------
//
//IDENT:       AUTOR:              DEPT:                           DATE:
//
//FC3.2.0      A.Egli              CT3                            06-Jan-2005
//              Code10: Control DirectCtrlLC (DB10)
//              Code12: LCDone (DB10)
//FC3.1.3      A.Egli              CT3                            13-Jun-2002
//              FCDone: Reset VarAnswerTime for PC 1 to 4
//FC3.1.2      A.Egli              CT3                            22-Mai-2002
//              FCDone: Reset VarAnswerTime
//FC3.1.1      A.Egli              CT3                             5-Feb-2002
//              Field DB3.GC.Revision: Is set to -1 in methode FcExamine
//FC3.1A       A.Egli              AEE61                           5-Jun-96
//              1st Release
//
//-------------------------------------------------------------------------
//
//PURPOSE:     MANUAL : ....... .DOC
//             
//
//RESTRICTIONS:
//
//-------------------------------------------------------------------------
//
//
AUTHOR : EA
FAMILY : GCS7SYS
NAME : PCD_Main
VERSION : 2.0
VAR_TEMP
  Code : INT ;
  Len : INT ;
  tmpByteNr : INT ;
  tmpFault : BOOL ;
  tmpBytePara : INT ;
  tmpDBSource : INT ;
  BitNr : INT ;
  tmpErrCode : INT ;
  tmpDBLen : WORD ;
  tmpWrite : BOOL ;
  tmpLen : INT ;
  tmpLenClear : DWORD ;
END_VAR
BEGIN
NETWORK
TITLE = Save
      T     #Code;	// Code
NETWORK
TITLE = FcControl: Code=0
//Control is interface to long locked (ParAnswerTime)
//
      L     #Code;
      L     0;
      <>I;
      JC    F1;
      L     "SYS_DirectCtrlDB".PC.Hsk;	//PC.Hsk
      <>I;
      JC    X2;
      T     "SYS_DirectCtrlDB".VarAnswerTime;	//VarAnswerTime
      BEU;
//== Test Read DB
X2:   L     860;	// ObjectType=DB
      L     "SYS_DirectCtrlDB".PC.ObjectType;	//ObjectType
      <>I;
      JC    X2c;
//- Test if DB existis
      CALL  "SYS_Copy_DBtoDB" (
           DBSource                 := "SYS_DirectCtrlDB".PC.ObjectNo,
           ByteSource               := 0,
           DBDest                   := 3,
           ByteDest                 := 20,
           NoOfByte                 := 1,
           Fault                    := #tmpFault);
      A     #tmpFault;
      JC    aX3;
      L     "SYS_DirectCtrlDB".PC.ObjectNo;
      T     #tmpDBSource;
      OPN   DI [#tmpDBSource];
      L     "SYS_DirectCtrlDB".PC.Value[2];	//Len in Byte
      T     #tmpLen;
      L     "SYS_DirectCtrlDB".PC.Value[1];	//FirstByte
      T     #tmpByteNr;
      L     "SYS_DirectCtrlDB".PC.Value[2];
      +I;
      L     DILG;
      <=I;
      JC    aX3a;
      L     "SYS_DirectCtrlDB".PC.Value[1];	//First Byte
      -I;
      T     #tmpLen;
      T     "SYS_DirectCtrlDB".PC.Value[2];	//Len in Byte
aX3a: AN    "SYS_DirectCtrlDB".PC.Hsk.FDefinePara;
      JC    exam;
      CALL  "SYS_Copy_DBtoDB" (
           DBSource                 := 3,
           ByteSource               := 62,
           DBDest                   := "SYS_DirectCtrlDB".PC.ObjectNo,
           ByteDest                 := #tmpByteNr,
           NoOfByte                 := #tmpLen,
           Fault                    := #tmpFault);
      JU    ini;
exam: L     P#DBX 62.0;
      T     #tmpLenClear;
loCr: L     0;
      T     DBD [#tmpLenClear];
      L     #tmpLenClear;
      L     P#4.0;
      +D;
      T     #tmpLenClear;
      L     P#DBX 252.0;
      <=D;
      JC    loCr;
      CALL  "SYS_Copy_DBtoDB" (
           DBSource                 := "SYS_DirectCtrlDB".PC.ObjectNo,
           ByteSource               := #tmpByteNr,
           DBDest                   := 3,
           ByteDest                 := 62,
           NoOfByte                 := #tmpLen,
           Fault                    := #tmpFault);
ini:  SET;
      S     "SYS_DirectCtrlDB".ChangeBit.CBit1;
      L     0;
      T     "SYS_DirectCtrlDB".PC.Hsk;
      T     "SYS_DirectCtrlDB".PC.ErrCode;
      T     "SYS_DirectCtrlDB".PC.ErrObj;
      T     "SYS_DirectCtrlDB".VarAnswerTime;
      BEU;	//CBitWrite
X2c:  L     0;
      L     "SYS_DirectCtrlDB".ParAnswerTime;	//Hsk
      <I;	//->PC.ErrCode
      JC    aOK2;	//->PC.ErrCode
      L     1;	//--> VarAnswerTime
aOK2: L     "SYS_DirectCtrlDB".VarAnswerTime;
//===================================
      <I;
      JC    aX3;	//ParAnswerTime
      +     1;
      T     "SYS_DirectCtrlDB".VarAnswerTime;
      BEU;	//Init: ParAnswerTime
aX3:  L     0;	//VarAnswerTime
      T     DB3.DBW 9;
      L     21;
      T     "SYS_DirectCtrlDB".PC.ErrCode;
      L     0;	//--> VarAnswerTime
      T     "SYS_DirectCtrlDB".PC.Hsk;	//=== error ===================
      S     "SYS_DirectCtrlDB".ChangeBit.CBit1;
      BEU;	//--> VarAnswerTime
NETWORK
TITLE = FcExamine : Code=1
//Copy datas from object to PcControl DB
//
//Input: InDynAddr: 1st byte of dynamic data
//       InDynLen : length of dynamic data in byte
//       InParaAddr: 1st byte of parameter
//       InParaLen : length of parameter in byte
//
F1:   L     1;
      L     #Code;
      <>I;
      JC    F2;
//--- Copy Dynamic Datas
      L     DINO;
      T     #tmpDBSource;
      T     "SYS_DirectCtrlDB".GC.InDBNr;
      L     DW#16#FFFFF;
      L     "SYS_DirectCtrlDB".GC.InDynAddr;	//GC.InDynAddr
      AD;
      SRD   3;
      T     #tmpByteNr;
      CALL  "SYS_Copy_DBtoDB" (
           DBSource                 := #tmpDBSource,
           ByteSource               := #tmpByteNr,
           DBDest                   := 3,
           ByteDest                 := 58,
           NoOfByte                 := "SYS_DirectCtrlDB".GC.InDynLen,
           Fault                    := #tmpFault);	//DB3 / GC.InDynLen
//--- Copy Parameters
      L     DW#16#FFFFFF;
      L     "SYS_DirectCtrlDB".GC.InParaAddr;	//GC.InParAddr
      AD;
      SRD   3;
      T     #tmpByteNr;
      L     "SYS_DirectCtrlDB".GC.InDynLen;	//GC.InDynLen
      +     58;
      T     #tmpBytePara;
      CALL  "SYS_Copy_DBtoDB" (
           DBSource                 := #tmpDBSource,
           ByteSource               := #tmpByteNr,
           DBDest                   := 3,
           ByteDest                 := #tmpBytePara,
           NoOfByte                 := "SYS_DirectCtrlDB".GC.InParaLen,
           Fault                    := #tmpFault);	//DB3 / GC.InParLen
      L     -1;
      T     "SYS_DirectCtrlDB".GC.Revision;
      JU    Done;
NETWORK
TITLE = FcDone
F2:   L     2;
      L     #Code;
      <>I;
      JC    F5;
Done: L     "SYS_DirectCtrlDB".PC.Hsk;	//Ksk
      L     0;
      ==I;
      BEC;
      S     "SYS_DirectCtrlDB".ChangeBit.CBit1;	//CBitWrite
      T     "SYS_DirectCtrlDB".PC.Hsk;	//Hsk
      T     "SYS_DirectCtrlDB".PC.ErrCode;	//->PC.ErrCode
      T     "SYS_DirectCtrlDB".PC.ErrObj;	//->PC.ErrCode
      T     "SYS_DirectCtrlDB".VarAnswerTime;	//[1.2]
      BEU;
NETWORK
TITLE = FcControlPC1to4 : Code 5
//DB by call = Actual Control DB of PC
//
F5:   L     5;
      L     #Code;
      <>I;
      JC    F10;
      CDB;	//Instanz DB = Actual Control DB
      L     DIW 42;	//CtrDB.PC.Hsk
      L     0;
      <>I;
      JC    dX2;
      T     DIW 18;	//CtrDB.VarAnswerTime
      JU    dOK;
dX2:  L     0;
      L     DIW 14;	//CtrDB.ParAnswerTime
      <I;
      JC    dOK2;
      L     1;	//Init:ParAnswerTime
dOK2: L     DIW 18;	//CtrDB.VarAnswerTime
      <I;
      JC    dERR;
      +     1;
      T     DIW 18;	// --> CtrDB.VarAnswerTime
      JU    dOK;	// === error ===================
dERR: L     0;	// 
      T     DIW 18;	// --> CtrDB.VarAnswerTime
      L     22;	// Illegal object
      T     DIW 46;	// ->err_code
      L     0;	//  
      T     DIW 42;	// ->CtrDB.Hsk
// === Handshake with DB3 ======
dOK:  L     DIW 42;	// CtrDB.Hsk
      L     0;	// 
      ==I;	// 
      JC    dTST;	// 
      L     "SYS_DirectCtrlDB".PC.Hsk;	// DB3.Hsk
      L     0;	// 
      <>I;	// 
      BEC;	// -->locked
      A     "SYS_DirectCtrlDB".ChangeBit.CBit1;	// DB3.CBit1
      JC    dTST;
//=== Move data to DB3 ===============
      L     DINO;
      T     #tmpDBSource;
      CALL  "SYS_Copy_DBtoDB" (
           DBSource                 := #tmpDBSource,
           ByteSource               := 42,
           DBDest                   := 3,
           ByteDest                 := 42,
           NoOfByte                 := 216,
           Fault                    := #tmpFault);	// DB3 / GC.InDynLen
      L     DINO;
      T     "SYS_DirectCtrlDB".VarActControlDB;	//VarActControlDB
      BEU;
//=== Read data back from DB 3 =====
dTST: L     DINO;
      L     "SYS_DirectCtrlDB".VarActControlDB;	//DB3.VarActControlDB
      <>I;
      A(;
      L     0;
      <>I;
      );
      ON    "SYS_DirectCtrlDB".ChangeBit.CBit1;	//DB3.CBit1
      BEC;
      L     DINO;
      T     #tmpDBSource;
      CALL  "SYS_Copy_DBtoDB" (
           DBSource                 := 3,
           ByteSource               := 20,
           DBDest                   := #tmpDBSource,
           ByteDest                 := 20,
           NoOfByte                 := 238,
           Fault                    := #tmpFault);	//Copy back include handshake / DB3 / DB3
      L     0;	//[1.3]
      T     DIW 18;	//CtrDB.VarAnswerTime       [1.3]
      A     "SYS_DirectCtrlDB".ChangeBit.CBit1;	//DB3.CBit1
      R     "SYS_DirectCtrlDB".ChangeBit.CBit1;	//DB3.CBit1
      S     DIX 41.0;	//CtrDB.CBit1
      BEU;
NETWORK
TITLE = FcControlLC: Code=10
//Control is interface to long locked (ParAnswerTime)
//
F10:  L     #Code;
      L     10;
      <>I;
      JC    F12;
      L     0;
      L     "SYS_DirectCtrlLCDB".PC.Hsk;	//PC.Hsk
      <>I;
      JC    F10A;
      T     "SYS_DirectCtrlLCDB".VarAnswerTime;	//VarAnswerTime
      BEU;
//== Test Read DB
F10A: L     0;
      L     "SYS_DirectCtrlLCDB".ParAnswerTime;	//Hsk
      <I;	//->PC.ErrCode
      JC    F10B;	//->PC.ErrCode
      L     1;	//--> VarAnswerTime
F10B: L     "SYS_DirectCtrlLCDB".VarAnswerTime;
//===================================
      <I;
      JC    F10C;	//ParAnswerTime
      AN    "SYS_Tick1s";
      BEC;
      +     1;
      T     "SYS_DirectCtrlLCDB".VarAnswerTime;
      BEU;	//Init: ParAnswerTime
F10C: L     0;	//VarAnswerTime
      T     "SYS_DirectCtrlLCDB".VarAnswerTime;
      L     21;
      T     "SYS_DirectCtrlLCDB".PC.ErrCode;
      L     0;	//--> VarAnswerTime
      T     "SYS_DirectCtrlLCDB".PC.Hsk;	//=== error ===================
      S     "SYS_DirectCtrlLCDB".ChangeBit.CBit1;
      BEU;	//--> VarAnswerTime
NETWORK
TITLE = [2.0] LCDone
F12:  L     12;
      L     #Code;
      <>I;
      JC    F13;
      L     "SYS_DirectCtrlLCDB".PC.Hsk;	//Ksk
      L     0;
      ==I;
      BEC;
      R     "SYS_DirectCtrlLCDB".GC.Set11Done;
      S     "SYS_DirectCtrlLCDB".ChangeBit.CBit1;	//CBitWrite
      T     "SYS_DirectCtrlLCDB".PC.Hsk;	//Hsk
      T     "SYS_DirectCtrlLCDB".PC.ErrCode;	//->PC.ErrCode
      T     "SYS_DirectCtrlLCDB".PC.ErrObj;	//->PC.ErrCode
      T     "SYS_DirectCtrlLCDB".VarAnswerTime;	//[1.2]
      BEU;
NETWORK
TITLE = END
F13:  NOP   0;
END_FUNCTION

FUNCTION "SYS_Horn_Code" : VOID	// FC 4
TITLE = Horn Modul
//COPYRIGHT:    (C) 2000 BUHLER AG, CH-9240 UZWIL  SWITZERLAND
//
//PRODUCT:      GCS7
//
//TITLE:        HornCode: Switch on horn 
//              
//
//--------------------------------------------------------------------------------
//
//IDENT:        AUTHOR:             DEPT:                              DATE:
//
//P01_FC004.1.0 A_Egli              CT3                                29.Okt.2002
//              1st Release
//
//--------------------------------------------------------------------------------
//
//PURPOSE: 
//
//REFERENCES: GCSOSMAN
//
//RESTRICTIONS: 
//
//--------------------------------------------------------------------------------
//
//InCode:
//------
//InCode=0 =Main Function Cylic Function
//InCode=1 =Main Function Coldstart/Newstart
//InCode=2 =Main Function Warm Start
//
AUTHOR : EA
FAMILY : ASW
NAME : HornCode
VERSION : 0.0
VAR_INPUT
  FcCode : INT ;	//Function Code: 1=Set Alarm , 2=Check StartWarning
  ParObjectType : INT ;	//Object Type of the calling Object
  ParObjectNo : INT ;	//Object number of the calling Object
  ParHornCode : INT ;	//HornCode of the calling object
END_VAR
VAR_TEMP
  tmpFlag : BOOL ;
  tmpHornCode : INT ;
END_VAR
BEGIN
NETWORK
TITLE = StartWarning
      L     #FcCode;
      L     0;
      <>I;
      JC    ALJ0;
//===============================
//1-A901Horn : Alarmhorn 1
//===============================
      CLR;
      O     DB100.DBX 36.0;
      O     DB100.DBX 46.0;
      =     "SYS_HornDB"._1_A901Horn.StartWarning;
      A     "SYS_HornDB".All.CmdHornOff;
      S     "SYS_HornDB"._1_A901Horn.CmdHornOff;
//===============================
//1-A902Horn : Alarmhorn 2
//===============================
      CLR;
      O     DB100.DBX 56.0;
      O     DB100.DBX 66.0;
      =     "SYS_HornDB"._1_A902Horn.StartWarning;
      A     "SYS_HornDB".All.CmdHornOff;
      S     "SYS_HornDB"._1_A902Horn.CmdHornOff;
//===============================
//1-A903Horn : Alarmhorn 3
//===============================
      CLR;
      O     DB100.DBX 76.0;
      O     DB100.DBX 86.0;
      =     "SYS_HornDB"._1_A903Horn.StartWarning;
      A     "SYS_HornDB".All.CmdHornOff;
      S     "SYS_HornDB"._1_A903Horn.CmdHornOff;
//===============================
//1-A904Horn : Alarmhorn 4
//===============================
      CLR;
      O     DB100.DBX 96.0;
      O     DB100.DBX 106.0;
      =     "SYS_HornDB"._1_A904Horn.StartWarning;
      A     "SYS_HornDB".All.CmdHornOff;
      S     "SYS_HornDB"._1_A904Horn.CmdHornOff;
//===============================
//Init Flag
//===============================
      A     "SYS_HornDB".All.CmdHornOff;
      R     "SYS_HornDB".All.CmdHornOff;
      BEU;
NETWORK
TITLE = FcCode=1: Subroutine Alarm
ALJ0: L     #FcCode;
      L     1;
      <>I;
      BEC;
NETWORK
TITLE =  HornCode = 1
      L     #ParHornCode;
      L     1;
      ==I;
      S     "SYS_HornDB"._1_A901Horn.CmdHornOn;
NETWORK
TITLE =  HornCode = 2
      L     #ParHornCode;
      L     2;
      ==I;
      S     "SYS_HornDB"._1_A901Horn.CmdHornOn;
NETWORK
TITLE =  HornCode = 4
      L     #ParHornCode;
      L     4;
      ==I;
      S     "SYS_HornDB"._1_A902Horn.CmdHornOn;
NETWORK
TITLE =  HornCode = 13
      L     #ParHornCode;
      L     13;
      ==I;
      =     #tmpFlag;
NETWORK
TITLE =  HornCode = 33
      L     #ParHornCode;
      L     33;
      ==I;
      =     #tmpFlag;
NETWORK
TITLE = End of Block
END_FUNCTION

FUNCTION "SYS_CallGroup" : VOID	// FC 9
TITLE = Call Groups
//COPYRIGHT:    (C) 1997 BY  BUHLER LTD.
//                           CH-9240 UZWIL  SWITZERLAND
//
//PRODUCT:      GCS7
//
//TITLE:        Aufruf Gruppen
//              Call Groups
//
//-------------------------------------------------------------------------
//
//IDENT:        AUTHOR:             DEPT:             DATE:
//
//FC009.1A      A_Egli              AEE61             28-Jan-98
//              1st Release
//
//-------------------------------------------------------------------------
//
//PURPOSE:      MANUAL : GCSOSMAN
//
//RESTRICTIONS:
//
//-------------------------------------------------------------------------
//
AUTHOR : EA
FAMILY : ASW
NAME : DEF
VERSION : 0.0
BEGIN
NETWORK
TITLE =
END_FUNCTION

FUNCTION "SYS_CallLineSection" : VOID	// FC 11
TITLE = Call Line Control
//COPYRIGHT:    (C) 1997 BY  BUHLER LTD.
//                           CH-9240 UZWIL  SWITZERLAND
//
//PRODUCT:      GCS90
//
//TITLE:        Aufruf Sektionssteuerungen Demo PIC
//              Call section control Demo PIC
//
//-------------------------------------------------------------------------
//
//IDENT:        AUTHOR:             DEPT:             DATE:
//
//FC011.1A      A_Egli              AEE61             14-Aug-97
//              1st Release
//
//-------------------------------------------------------------------------
//
//PURPOSE:      MANUAL : GCSOSMAN
//
//RESTRICTIONS: 
//
//-------------------------------------------------------------------------
//
NAME : PICDEMO
VERSION : 0.0
BEGIN
NETWORK
TITLE =
NETWORK
TITLE = Call Group control
NETWORK
TITLE = Call Methode Scale Control
END_FUNCTION

FUNCTION "TEST_IOSIMULI_Copy" : VOID	// FC 16
TITLE = Copy IO Manager
//COPYRIGHT:          (C) 1994 BY  BUHLER LTD.
//                                 CH-9240 UZWIL  SWITZERLAND
//
//PRODUCT:            GCS90 Obere Schichten
//
//TITLE:              Simulation of elements
// 
//-------------------------------------------------------------------
//
//IDENT:       AUTOR:              DEPT:             DATE:
//
//FC016.1B     EA                  CT3               25-Okt-99
//              Mit OB122 
//FC016.1A     EA                  CT3               14-Apr-97
//              1st Release
//
//-------------------------------------------------------------------
//
//PURPOSE:      
//
//RESTRICTIONS:
//
//-------------------------------------------------------------------
//
//
AUTHOR : EA
FAMILY : GCS90
NAME : SIMU
VERSION : 0.0
VAR_INPUT
  BlockCopy : BOOL ;
  CallSFC36 : BOOL ;	//Nur falls nicht OB122 eingesetzt wird
  LastIOByte : INT ;	//Länge Prozessabbild in Byte
END_VAR
VAR_TEMP
  tmpAddr : DINT ;
  tmpLastIOAddr : DWORD ;
END_VAR
BEGIN
NETWORK
TITLE =
      AN    #CallSFC36;
      JC    X1;
      CALL  "SIEMENS_MSK_FLT" (
           PRGFLT_SET_MASK          := DW#16#0,
           ACCFLT_SET_MASK          := DW#16#3F,
           RET_VAL                  := MW 250,
           PRGFLT_MASKED            := MD 248,
           ACCFLT_MASKED            := MD 252);
X1:   NOP   0;
NETWORK
TITLE =
      L     #LastIOByte;
      SLD   3;
      T     #tmpLastIOAddr;
NETWORK
TITLE = Copy Output
      AN    #BlockCopy;
      JC    O1;
      CALL  "SIEMENS_BLKMOV" (
           SRCBLK                   := P#Q 0.0 BYTE 128,
           RET_VAL                  := MW 200,
           DSTBLK                   := P#DB17.DBX 0.0 BYTE 128);
      L     #LastIOByte;
      L     128;
      <I;
      JC    I0;
      CALL  "SIEMENS_BLKMOV" (
           SRCBLK                   := P#Q 128.0 BYTE 128,
           RET_VAL                  := MW 200,
           DSTBLK                   := P#DB17.DBX 128.0 BYTE 128);
      L     #LastIOByte;
      L     256;
      <I;
      JC    I0;
      CALL  "SIEMENS_BLKMOV" (
           SRCBLK                   := P#Q 256.0 BYTE 128,
           RET_VAL                  := MW 200,
           DSTBLK                   := P#DB17.DBX 256.0 BYTE 128);
      L     #LastIOByte;
      L     384;
      <I;
      JC    I0;
      CALL  "SIEMENS_BLKMOV" (
           SRCBLK                   := P#Q 384.0 BYTE 128,
           RET_VAL                  := MW 200,
           DSTBLK                   := P#DB17.DBX 384.0 BYTE 128);
      JU    I0;
O1:   NOP   0;
      OPN   "TEST_IOSimuliOutput";
      L     P#0.0;
      T     #tmpAddr;
o2:   L     QW [#tmpAddr];
      T     DBW [#tmpAddr];
      L     #tmpAddr;
      +     L#16;
      T     #tmpAddr;
      L     #tmpLastIOAddr;
      <=D;
      JC    o2;
NETWORK
TITLE = Copy Input
I0:   NOP   0;
      AN    #BlockCopy;
      JC    i1;
      CALL  "SIEMENS_BLKMOV" (
           SRCBLK                   := P#DB16.DBX 0.0 BYTE 128,
           RET_VAL                  := MW 200,
           DSTBLK                   := P#I 0.0 BYTE 128);
      L     #LastIOByte;
      L     128;
      <I;
      JC    I0;
      CALL  "SIEMENS_BLKMOV" (
           SRCBLK                   := P#DB16.DBX 128.0 BYTE 128,
           RET_VAL                  := MW 200,
           DSTBLK                   := P#I 128.0 BYTE 128);
      L     #LastIOByte;
      L     256;
      <I;
      JC    I0;
      CALL  "SIEMENS_BLKMOV" (
           SRCBLK                   := P#DB16.DBX 256.0 BYTE 128,
           RET_VAL                  := MW 200,
           DSTBLK                   := P#I 256.0 BYTE 128);
      L     #LastIOByte;
      L     384;
      <I;
      JC    I0;
      CALL  "SIEMENS_BLKMOV" (
           SRCBLK                   := P#DB16.DBX 384.0 BYTE 128,
           RET_VAL                  := MW 200,
           DSTBLK                   := P#I 384.0 BYTE 128);
      BEU;
i1:   OPN   "TEST_IOSimuliInput";
      L     P#0.0;
      T     #tmpAddr;
i2:   L     DBW [#tmpAddr];
      T     IW [#tmpAddr];
      L     #tmpAddr;
      +     L#16;
      T     #tmpAddr;
      L     #tmpLastIOAddr;
      <=D;
      JC    i2;
END_FUNCTION

FUNCTION "GCS7_TON_LONG" : VOID	// FC 17
TITLE = Timer  TON
//COPYRIGHT:    (C) 1998 BY  BUHLER AG
//                           CH-9240 UZWIL  SWITZERLAND
//
//PRODUCT:      GCS7
//
//TITLE:        Timer TON long
//              
//
//-------------------------------------------------------------------------
//
//IDENT:        AUTHOR:             DEPT:             DATE:
//
//FC17.1A       A.Egli              CT3               12-Feb-2003
//              1st Release
//
//-------------------------------------------------------------------------
//
//PURPOSE: 
//
//RESTRICTIONS: 
//
//-------------------------------------------------------------------------
//
//Functions
//=========
//
AUTHOR : EA
FAMILY : ASW
NAME : TON
VERSION : 1.0
VAR_INPUT
  IN : BOOL ;	//EnableTimer
  PT : DINT ;	//Timer Value Target [0.1s]
END_VAR
VAR_OUTPUT
  Q : BOOL ;	//Delay Done
END_VAR
VAR_IN_OUT
  ET : DINT ;	//Actual Value Timer [0.1s]
END_VAR
BEGIN
NETWORK
TITLE = Initialisation
      A     #IN;
      JC    aEnd;
      L     #PT;
      T     #ET;
aEnd: NOP   0;
NETWORK
TITLE =
      AN    "GCS7_Gr_OutTick200ms";
      ON    #IN;
      JC    bNot;
      L     #ET;
      L     L#2;
      -D;
      JP    bVal;
      L     L#0;
bVal: T     #ET;
bNot: L     L#0;
      L     #ET;
      >=D;
      A     #IN;
      =     #Q;
END_FUNCTION

FUNCTION "GCS7_TON" : VOID	// FC 18
TITLE = Timer  TON
//COPYRIGHT:    (C) 1998 BY  BUHLER AG
//                           CH-9240 UZWIL  SWITZERLAND
//
//PRODUCT:      GCS7
//
//TITLE:        Timer TON
//              
//
//-------------------------------------------------------------------------
//
//IDENT:        AUTHOR:             DEPT:             DATE:
//
//FC18.1A       A.Egli              CT3               12-Feb-2003
//              1st Release
//
//-------------------------------------------------------------------------
//
//PURPOSE: 
//
//RESTRICTIONS: 
//
//-------------------------------------------------------------------------
//
//Functions
//=========
//
AUTHOR : EA
FAMILY : ASW
NAME : TON
VERSION : 1.0
VAR_INPUT
  IN : BOOL ;	//EnableTimer
  PT : INT ;	//Timer Value Target [0.1s]
END_VAR
VAR_OUTPUT
  Q : BOOL ;	//Delay Done
END_VAR
VAR_IN_OUT
  ET : INT ;	//Actual Value Timer [0.1s]
END_VAR
BEGIN
NETWORK
TITLE = Initialisation
      A     #IN;
      JC    aEnd;
      L     #PT;
      T     #ET;
aEnd: NOP   0;
NETWORK
TITLE =
      AN    "GCS7_Gr_OutTick200ms";
      ON    #IN;
      JC    bNot;
      L     #ET;
      L     2;
      -I;
      JP    bVal;
      L     0;
bVal: T     #ET;
bNot: L     0;
      L     #ET;
      >=I;
      A     #IN;
      =     #Q;
END_FUNCTION

FUNCTION "SYS_Analog_S5_to_S7" : VOID	// FC 19
TITLE = Scale S7 Analogues for S5
//COPYRIGHT:    (C) 1998 BY  BUHLER AG
//                           CH-9240 UZWIL  SWITZERLAND
//
//PRODUCT:      AME01_98
//
//TITLE:        Scale S7 Analogues for S5
//              
//
//-------------------------------------------------------------------------
//
//IDENT:        AUTHOR:             DEPT:             DATE:
//
//FC105.1A      GS                  CDDP              15-Jan-2000
//              1st Release
//
//-------------------------------------------------------------------------
//
//PURPOSE: 
//
//RESTRICTIONS: 
//
//-------------------------------------------------------------------------
//
//Functions
//=========
//
//  01 - S5 Analogue Input 0..20mA
//  02 - S5 Analogue Input 4..20mA
//  03 - S5 Analogue Output 0..20mA or 4..20mA card
//  04 - S5 Analogue Output 4..20mA on a 0..20mA card
//
//
AUTHOR : GS
FAMILY : ASW
NAME : ANA_S5_S
VERSION : 1.0
VAR_INPUT
  function_no : INT ;	//function selection
END_VAR
VAR_TEMP
  Inputvalue : INT ;
  OutputValue : INT ;
END_VAR
BEGIN
NETWORK
TITLE = Initialisation
      TAK;
      T     #Inputvalue;
NETWORK
TITLE = S5 Analogue Input 0..20mA
// (network holds code this reader does not know; not shown)
// S5 Analogue inputs cards 0..20mA give a number of 0..2048
// Bottom 3 bits are used for over/under range indication from the card
// All S7 modules use 0..27648 as 0..100%
// Conversion formula is:-
//  
//     S5Value  * 27648
//     -------
//      2048
// 
NETWORK
TITLE = S5 Analogue Input 4..20mA
// (network holds code this reader does not know; not shown)
// S5 Analogue inputs cards 4..20mA give a number of 0..2560
// but have an offset of 512. This gives 512..2560 = 4..20mA
// 2048 units cover 16mA.
// Bottom 3 bits are used for over/under range indication from the card
// All S7 modules use 0..27648 as 0..100%
// Conversion formula is:-
//  
//     (S5Value - 512)  * 27648
//     ---------------
//          2048
// 
NETWORK
TITLE = S5 Analogue Output 0..20mA or 4..20mA card
      L     #function_no;
      L     3;
      <>I;
      JC    en03;
// S5 Analogue Outputs cards use a number of 0..1024
// Bottom 4 bits are not used used
// All S7 modules use 0..27648 as 0..100%
// Conversion formula is:-
//  
//     S7Value  * 1024
//     -------
//      27648
// 
      L     #Inputvalue;
      DTR;
      L     2.764800e+04;	// 27648
      /R;
      L     1.024000e+03;	// 1024
      *R;
      RND;
      SLW   4;
      T     #OutputValue;
en03: NOP   0;
NETWORK
TITLE = S5 Analogue Output 4..20mA on a 0..20mA card
      L     #function_no;
      L     4;
      <>I;
      JC    en04;
// S5 Analogue Outputs cards use a number of 0..1024
// Bottom 4 bits are not used used
// All S7 modules use 0..27648 as 0..100%
// Conversion formula is:-
//  
//    ( S7Value  * 820 ) + 204
//      -------
//       27648
// 
// Note:   820 is 4/5ths of 1024    (for the 4..20mA portion)
//         204 is 1/5th of 1024     (for the 0..4mA portion)
// 
      L     #Inputvalue;
      DTR;
      L     2.764800e+04;	// 27648
      /R;
      L     8.200000e+02;	// 820
      *R;
      L     2.040000e+02;	// 204
      +R;
      RND;
      SLW   4;
      T     #OutputValue;
en04: NOP   0;
NETWORK
TITLE = Output final value
      L     #OutputValue;
END_FUNCTION

FUNCTION "CWA_ScaleSimul" : VOID	// FC 39
TITLE = CWA SCALE SIMULATION
//
//COPYRIGHT:    (C) 1996 BY  BUHLER LTD.
//                           CH-9240 UZWIL  SWITZERLAND
//
//PRODUCT:      CWA
//
//TITLE:        SCALE CONTROL: SCALE SIMULATION
//
//-------------------------------------------------------------------------
//
//IDENT:        AUTOR:              DEPT:                         DATE:
//
//FC39.2.1      A. Egli            CT3                            06-Nov-2004
//              Negative Weighing: Invert Flowrate when slow dosing
//FC39.2.0      A. Egli            CT3                            26-Jun-2000
//              New release, without timer
//
//-------------------------------------------------------------------------
//
//PURPOSE:      MANUAL : CWAMAN
//
//RESTRICTIONS:
//
//-------------------------------------------------------------------------
//
//$EJECT
//
AUTHOR : EA
FAMILY : CWA
NAME : CWASim
VERSION : 2.1
VAR_INPUT
  Reset : BOOL ;	//Reset weight
  Refill : BOOL ;	//1= Refill doubt
  ErrorFill : BOOL ;	//Error Filling
  ErrorEmpty : BOOL ;	//Error Emptying
  ParIntervall : INT ;	//Calling intervall (ms)
  ParFlowrateFastDos : DINT ;	//Flowrate at fast dosing (gr/s)
  ParFlowrateSlowDos : DINT ;	//Flowrate at slow dosing (gr/s)
  ParFlowrateEmptying : DINT ;	//Flowrate emptying/refill (gr/s)
  ParDlyFastDos : INT ;	//Switch off delay fast Dosing [ms]
  ParDlySlowDos : INT ;	//Switch off delay slow Dosing [ms]
END_VAR
VAR_IN_OUT
  InOutTimerValue1 : INT ;	//Internal used
  InOutTimerValue2 : INT ;	//Internal used
  InOutDeltaWeight : REAL ;	//Internal used [kg]
END_VAR
VAR_TEMP
  tmpFlowrate : DINT ;
  tmpDosing : BOOL ;
  tmpDosingFast : BOOL ;
  tmpDigits : DINT ;
  tmpScaleUnit : REAL ;
END_VAR
BEGIN
NETWORK
TITLE = FC-PARAMETER
//
//
//ACTUAL DB BY CALL: SCALE DB
//
//
NETWORK
TITLE = Timer
      L     0;
      T     #tmpFlowrate;
      L     0;
      L     #InOutTimerValue1;
      >=I;
      JC    I2;
      L     #ParIntervall;
      -I;
      T     #InOutTimerValue1;
I2:   L     0;
      L     #InOutTimerValue2;
      >=I;
      JC    I3;
      L     #ParIntervall;
      -I;
      T     #InOutTimerValue2;
I3:   NOP   0;
NETWORK
TITLE = Reset
      AN    #Reset;
      JC    RJ0;
      L     0;
      T     DBD 148;	// --> "CWA01".ME.VarScaleValueInput
      T     #InOutTimerValue1;
      T     #InOutTimerValue2;
      BEU;
RJ0:  NOP   0;
NETWORK
TITLE = Refill
      AN    DBX 251.4;	//"CWA01".Status.StaRefillReq
      ON    #Refill;
      JC    RFJ0;
      L     #ParFlowrateEmptying;
      T     #tmpFlowrate;
      JU    CALC;
RFJ0: NOP   0;
NETWORK
TITLE = Emptying
      A     DBX 7.0;	//  "CWA01".ParScalceCfg1.ParNegWeighing 
      JC    EPJ0;
      A     DBX 54.5;	// "CWA01".ToCWA.InpClosed
      O     DBX 7.1;	// "CWA01".ParScalceCfg1.ParNoEmptying
      JC    EPJ0;
      L     DBD 254;
      L     DBD 180;	// "CWA01".ScalePara.ParEmptyWt
      <D;
      O     #ErrorEmpty;
      JC    CALC;
      L     #ParFlowrateEmptying;
      NEGD;
      T     #tmpFlowrate;
      JU    CALC;	//--> Calculate
EPJ0: NOP   0;
NETWORK
TITLE = Dosing
//===========================================
//=Switch off Delay Time
//===========================================
//Reconveying
      AN    DBX 248.1;	// "CWA01".Status.StaReconveying 
      JC    DFas;
      AN    DBX 42.7;	// "CWA01".ToASW.OutpDosing
      JC    DFas;
      L     200;	//[ms]
      T     #InOutTimerValue2;
      L     #ParFlowrateSlowDos;
      T     #tmpFlowrate;
      JU    DJ1;	//[2.1]
//===========================================
//Switch Off Delay Fast Dosing
DFas: AN    DBX 42.6;	// "CWA01".ToASW.OutpDosingFast
      JC    DSlo;
      L     #ParDlyFastDos;	// DelayFastDosing
      T     #InOutTimerValue1;
      L     #ParFlowrateFastDos;
      T     #tmpFlowrate;
      JU    DJ1;
//===========================================
//Switch Off Delay Slow Dosing
//===========================================
DSlo: AN    DBX 42.7;	// "CWA01".ToASW.OutpDosing
      JC    DDly;
      L     #ParDlySlowDos;	// DelaySlowDosing
      T     #InOutTimerValue2;
      L     1;
      >=I;
      JC    DDly;
      T     #InOutTimerValue2;
//==========================================
//Switch off delay
DDly: L     #InOutTimerValue1;
      L     0;
      >I;
      L     #ParFlowrateFastDos;
      T     #tmpFlowrate;
      JC    DJ1;
      L     #InOutTimerValue2;
      L     0;
      >I;
      L     #ParFlowrateSlowDos;
      T     #tmpFlowrate;
      JC    DJ1;
      L     0;
      T     #tmpFlowrate;
DJ1:  AN    DBX 7.0;	//"CWA01".ParScalceCfg1.ParNegWeighing
      JC    DJ0;
      L     #tmpFlowrate;
      NEGD;
      T     #tmpFlowrate;
DJ0:  NOP   0;
NETWORK
TITLE = Calculate delta weight
      A     #ErrorFill;
      O     DBX 244.2;	// "CWA01".Fault.EsReading
      JC    cJ0;
CALC: L     DBW 30;
      L     0;
      ==I;
      L     1.000000e+00;
      JC    cC1;
      L     DBW 30;
      L     1;
      ==I;
      L     1.000000e-01;
      JC    cC1;
      L     DBW 30;
      L     2;
      ==I;
      L     1.000000e-02;
      JC    cC1;
      L     1.000000e-03;
cC1:  T     #tmpScaleUnit;	//  [gr /1000]
      L     #ParIntervall;	//[ms]
      DTR;
      L     1.000000e+03;
      /R;	//-->[s]
      L     #tmpFlowrate;	// [gr/s]
      DTR;
      *R;
      L     1.000000e-03;
      *R;
      L     #tmpScaleUnit;
      /R;
      L     #InOutDeltaWeight;	//InOutDeltaWeight [kg]
      +R;
      T     #InOutDeltaWeight;	//InOutDeltaWeight [kg]
      L     DBD 126;
      /R;
      RND;
      T     #tmpDigits;
      L     0;
      ==D;
      JC    cJ0;
      L     #tmpDigits;
      DTR;
      L     DBD 126;
      *R;
      L     #InOutDeltaWeight;	//InOutDeltaWeight
      TAK;
      -R;
      T     #InOutDeltaWeight;	//InOutDeltaWeight
// Calculate value in digits
      L     DBD 148;	// "CWA01".ME.VarScaleValueInput
      L     #tmpDigits;
      +D;
      T     DBD 148;	// -->"CWA01".ME.VarScaleValueInput
//Scale weight >= 0
      L     0;
      >=D;
      JC    cJ0;
      T     DBD 148;	// "CWA01".ME.VarScaleValueInput
cJ0:  NOP   0;
NETWORK
TITLE = Simulate Alarm EsReading 
//========================
//Test maximum Value
      L     DBD 12;	// "CWA01".ParScaleCapacityWt
      +     L#30;	// +30
      L     DBD 254;	// "CWA01".ScaleWt
      <D;
      S     DBX 244.2;	// "CWA01".Fault.EsReading
// Test Minimum Value
      L     DBD 254;	// "CWA01".ScaleWt
      L     L#-30;
      <D;
      S     DBX 244.2;	// "CWA01".Fault.EsReading
NETWORK
TITLE =
      BE;
END_FUNCTION

